Fanuc TP program (LS listing): FM140311.ls

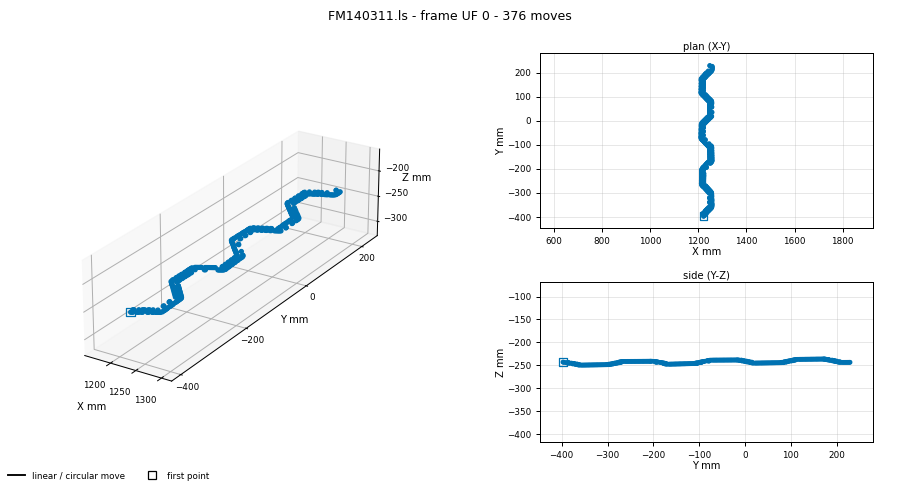
[picture p0: tool path of FM140311.ls in frame UF 0, 376 of 376 moves have a stored position in this frame; points joined in program order, loops and branches not executed]
/PROG  FM140311
/ATTR
OWNER		= MNEDITOR;
COMMENT		= "Auto FANUC move";
PROG_SIZE	= 0;
CREATE		= DATE 26-05-06  TIME 14:03:11;
MODIFIED	= DATE 26-05-06  TIME 14:03:11;
FILE_NAME	= ;
VERSION		= 0;
LINE_COUNT	= 381;
MEMORY_SIZE	= 0;
PROTECT		= READ_WRITE;
TCD:  STACK_SIZE	= 0,
      TASK_PRIORITY	= 50,
      TIME_SLICE	= 0,
      BUSY_LAMP_OFF	= 0,
      ABORT_REQUEST	= 0,
      PAUSE_REQUEST	= 0;
DEFAULT_GROUP	= 1,*,*,*,*;
CONTROL_CODE	= 00000000 00000000;
/MN
   1:  UFRAME_NUM=0 ;
   2:  UTOOL_NUM=1 ;
   3:  R[93]=10 ;
   4:  L P[1] 7mm/sec FINE ;
   5:  L P[2] 7mm/sec CNT50 ;
   6:  L P[3] 7mm/sec CNT50 ;
   7:  L P[4] 7mm/sec CNT50 ;
   8:  L P[5] 7mm/sec CNT50 ;
   9:  L P[6] 7mm/sec CNT50 ;
  10:  L P[7] 7mm/sec CNT50 ;
  11:  L P[8] 7mm/sec CNT50 ;
  12:  L P[9] 7mm/sec CNT50 ;
  13:  L P[10] 7mm/sec CNT50 ;
  14:  L P[11] 7mm/sec CNT50 ;
  15:  L P[12] 7mm/sec CNT50 ;
  16:  L P[13] 7mm/sec CNT50 ;
  17:  L P[14] 7mm/sec CNT50 ;
  18:  L P[15] 7mm/sec CNT50 ;
  19:  L P[16] 7mm/sec CNT50 ;
  20:  L P[17] 7mm/sec CNT50 ;
  21:  L P[18] 7mm/sec CNT50 ;
  22:  L P[19] 7mm/sec CNT50 ;
  23:  L P[20] 7mm/sec CNT50 ;
  24:  L P[21] 7mm/sec CNT50 ;
  25:  L P[22] 7mm/sec CNT50 ;
  26:  L P[23] 7mm/sec CNT50 ;
  27:  L P[24] 7mm/sec CNT50 ;
  28:  L P[25] 7mm/sec CNT50 ;
  29:  L P[26] 7mm/sec CNT50 ;
  30:  L P[27] 7mm/sec CNT50 ;
  31:  L P[28] 7mm/sec CNT50 ;
  32:  L P[29] 7mm/sec CNT50 ;
  33:  L P[30] 7mm/sec CNT50 ;
  34:  L P[31] 7mm/sec CNT50 ;
  35:  L P[32] 7mm/sec CNT50 ;
  36:  L P[33] 7mm/sec CNT50 ;
  37:  L P[34] 7mm/sec CNT50 ;
  38:  L P[35] 7mm/sec CNT50 ;
  39:  L P[36] 7mm/sec CNT50 ;
  40:  L P[37] 7mm/sec CNT50 ;
  41:  L P[38] 7mm/sec CNT50 ;
  42:  L P[39] 7mm/sec CNT50 ;
  43:  L P[40] 7mm/sec CNT50 ;
  44:  L P[41] 7mm/sec CNT50 ;
  45:  L P[42] 7mm/sec CNT50 ;
  46:  L P[43] 7mm/sec CNT50 ;
  47:  L P[44] 7mm/sec CNT50 ;
  48:  L P[45] 7mm/sec CNT50 ;
  49:  L P[46] 7mm/sec CNT50 ;
  50:  L P[47] 7mm/sec CNT50 ;
  51:  L P[48] 7mm/sec CNT50 ;
  52:  L P[49] 7mm/sec CNT50 ;
  53:  L P[50] 7mm/sec CNT50 ;
  54:  L P[51] 7mm/sec CNT50 ;
  55:  L P[52] 7mm/sec CNT50 ;
  56:  L P[53] 7mm/sec CNT50 ;
  57:  L P[54] 7mm/sec CNT50 ;
  58:  L P[55] 7mm/sec CNT50 ;
  59:  L P[56] 7mm/sec CNT50 ;
  60:  L P[57] 7mm/sec CNT50 ;
  61:  L P[58] 7mm/sec CNT50 ;
  62:  L P[59] 7mm/sec CNT50 ;
  63:  L P[60] 7mm/sec CNT50 ;
  64:  L P[61] 7mm/sec CNT50 ;
  65:  L P[62] 7mm/sec CNT50 ;
  66:  L P[63] 7mm/sec CNT50 ;
  67:  L P[64] 7mm/sec CNT50 ;
  68:  L P[65] 7mm/sec CNT50 ;
  69:  L P[66] 7mm/sec CNT50 ;
  70:  L P[67] 7mm/sec CNT50 ;
  71:  L P[68] 7mm/sec CNT50 ;
  72:  L P[69] 7mm/sec CNT50 ;
  73:  L P[70] 7mm/sec CNT50 ;
  74:  L P[71] 7mm/sec CNT50 ;
  75:  L P[72] 7mm/sec CNT50 ;
  76:  L P[73] 7mm/sec CNT50 ;
  77:  L P[74] 7mm/sec CNT50 ;
  78:  L P[75] 7mm/sec CNT50 ;
  79:  L P[76] 7mm/sec CNT50 ;
  80:  L P[77] 7mm/sec CNT50 ;
  81:  L P[78] 7mm/sec CNT50 ;
  82:  L P[79] 7mm/sec CNT50 ;
  83:  L P[80] 7mm/sec CNT50 ;
  84:  L P[81] 7mm/sec CNT50 ;
  85:  L P[82] 7mm/sec CNT50 ;
  86:  L P[83] 7mm/sec CNT50 ;
  87:  L P[84] 7mm/sec CNT50 ;
  88:  L P[85] 7mm/sec CNT50 ;
  89:  L P[86] 7mm/sec CNT50 ;
  90:  L P[87] 7mm/sec CNT50 ;
  91:  L P[88] 7mm/sec CNT50 ;
  92:  L P[89] 7mm/sec CNT50 ;
  93:  L P[90] 7mm/sec CNT50 ;
  94:  L P[91] 7mm/sec CNT50 ;
  95:  L P[92] 7mm/sec CNT50 ;
  96:  L P[93] 7mm/sec CNT50 ;
  97:  L P[94] 7mm/sec CNT50 ;
  98:  L P[95] 7mm/sec CNT50 ;
  99:  L P[96] 7mm/sec CNT50 ;
 100:  L P[97] 7mm/sec CNT50 ;
 101:  L P[98] 7mm/sec CNT50 ;
 102:  L P[99] 7mm/sec CNT50 ;
 103:  L P[100] 7mm/sec CNT50 ;
 104:  L P[101] 7mm/sec CNT50 ;
 105:  L P[102] 7mm/sec CNT50 ;
 106:  L P[103] 7mm/sec CNT50 ;
 107:  L P[104] 7mm/sec CNT50 ;
 108:  L P[105] 7mm/sec CNT50 ;
 109:  L P[106] 7mm/sec CNT50 ;
 110:  L P[107] 7mm/sec CNT50 ;
 111:  L P[108] 7mm/sec CNT50 ;
 112:  L P[109] 7mm/sec CNT50 ;
 113:  L P[110] 7mm/sec CNT50 ;
 114:  L P[111] 7mm/sec CNT50 ;
 115:  L P[112] 7mm/sec CNT50 ;
 116:  L P[113] 7mm/sec CNT50 ;
 117:  L P[114] 7mm/sec CNT50 ;
 118:  L P[115] 7mm/sec CNT50 ;
 119:  L P[116] 7mm/sec CNT50 ;
 120:  L P[117] 7mm/sec CNT50 ;
 121:  L P[118] 7mm/sec CNT50 ;
 122:  L P[119] 7mm/sec CNT50 ;
 123:  L P[120] 7mm/sec CNT50 ;
 124:  L P[121] 7mm/sec CNT50 ;
 125:  L P[122] 7mm/sec CNT50 ;
 126:  L P[123] 7mm/sec CNT50 ;
 127:  L P[124] 7mm/sec CNT50 ;
 128:  L P[125] 7mm/sec CNT50 ;
 129:  L P[126] 7mm/sec CNT50 ;
 130:  L P[127] 7mm/sec CNT50 ;
 131:  L P[128] 7mm/sec CNT50 ;
 132:  L P[129] 7mm/sec CNT50 ;
 133:  L P[130] 7mm/sec CNT50 ;
 134:  L P[131] 7mm/sec CNT50 ;
 135:  L P[132] 7mm/sec CNT50 ;
 136:  L P[133] 7mm/sec CNT50 ;
 137:  L P[134] 7mm/sec CNT50 ;
 138:  L P[135] 7mm/sec CNT50 ;
 139:  L P[136] 7mm/sec CNT50 ;
 140:  L P[137] 7mm/sec CNT50 ;
 141:  L P[138] 7mm/sec CNT50 ;
 142:  L P[139] 7mm/sec CNT50 ;
 143:  L P[140] 7mm/sec CNT50 ;
 144:  L P[141] 7mm/sec CNT50 ;
 145:  L P[142] 7mm/sec CNT50 ;
 146:  L P[143] 7mm/sec CNT50 ;
 147:  L P[144] 7mm/sec CNT50 ;
 148:  L P[145] 7mm/sec CNT50 ;
 149:  L P[146] 7mm/sec CNT50 ;
 150:  L P[147] 7mm/sec CNT50 ;
 151:  L P[148] 7mm/sec CNT50 ;
 152:  L P[149] 7mm/sec CNT50 ;
 153:  L P[150] 7mm/sec CNT50 ;
 154:  L P[151] 7mm/sec CNT50 ;
 155:  L P[152] 7mm/sec CNT50 ;
 156:  L P[153] 7mm/sec CNT50 ;
 157:  L P[154] 7mm/sec CNT50 ;
 158:  L P[155] 7mm/sec CNT50 ;
 159:  L P[156] 7mm/sec CNT50 ;
 160:  L P[157] 7mm/sec CNT50 ;
 161:  L P[158] 7mm/sec CNT50 ;
 162:  L P[159] 7mm/sec CNT50 ;
 163:  L P[160] 7mm/sec CNT50 ;
 164:  L P[161] 7mm/sec CNT50 ;
 165:  L P[162] 7mm/sec CNT50 ;
 166:  L P[163] 7mm/sec CNT50 ;
 167:  L P[164] 7mm/sec CNT50 ;
 168:  L P[165] 7mm/sec CNT50 ;
 169:  L P[166] 7mm/sec CNT50 ;
 170:  L P[167] 7mm/sec CNT50 ;
 171:  L P[168] 7mm/sec CNT50 ;
 172:  L P[169] 7mm/sec CNT50 ;
 173:  L P[170] 7mm/sec CNT50 ;
 174:  L P[171] 7mm/sec CNT50 ;
 175:  L P[172] 7mm/sec CNT50 ;
 176:  L P[173] 7mm/sec CNT50 ;
 177:  L P[174] 7mm/sec CNT50 ;
 178:  L P[175] 7mm/sec CNT50 ;
 179:  L P[176] 7mm/sec CNT50 ;
 180:  L P[177] 7mm/sec CNT50 ;
 181:  L P[178] 7mm/sec CNT50 ;
 182:  L P[179] 7mm/sec CNT50 ;
 183:  L P[180] 7mm/sec CNT50 ;
 184:  L P[181] 7mm/sec CNT50 ;
 185:  L P[182] 7mm/sec CNT50 ;
 186:  L P[183] 7mm/sec CNT50 ;
 187:  L P[184] 7mm/sec CNT50 ;
 188:  L P[185] 7mm/sec CNT50 ;
 189:  L P[186] 7mm/sec CNT50 ;
 190:  L P[187] 7mm/sec CNT50 ;
 191:  L P[188] 7mm/sec CNT50 ;
 192:  L P[189] 7mm/sec CNT50 ;
 193:  L P[190] 7mm/sec CNT50 ;
 194:  L P[191] 7mm/sec CNT50 ;
 195:  L P[192] 7mm/sec CNT50 ;
 196:  L P[193] 7mm/sec CNT50 ;
 197:  L P[194] 7mm/sec CNT50 ;
 198:  L P[195] 7mm/sec CNT50 ;
 199:  L P[196] 7mm/sec CNT50 ;
 200:  L P[197] 7mm/sec CNT50 ;
 201:  L P[198] 7mm/sec CNT50 ;
 202:  L P[199] 7mm/sec CNT50 ;
 203:  L P[200] 7mm/sec CNT50 ;
 204:  L P[201] 7mm/sec CNT50 ;
 205:  L P[202] 7mm/sec CNT50 ;
 206:  L P[203] 7mm/sec CNT50 ;
 207:  L P[204] 7mm/sec CNT50 ;
 208:  L P[205] 7mm/sec CNT50 ;
 209:  L P[206] 7mm/sec CNT50 ;
 210:  L P[207] 7mm/sec CNT50 ;
 211:  L P[208] 7mm/sec CNT50 ;
 212:  L P[209] 7mm/sec CNT50 ;
 213:  L P[210] 7mm/sec CNT50 ;
 214:  L P[211] 7mm/sec CNT50 ;
 215:  L P[212] 7mm/sec CNT50 ;
 216:  L P[213] 7mm/sec CNT50 ;
 217:  L P[214] 7mm/sec CNT50 ;
 218:  L P[215] 7mm/sec CNT50 ;
 219:  L P[216] 7mm/sec CNT50 ;
 220:  L P[217] 7mm/sec CNT50 ;
 221:  L P[218] 7mm/sec CNT50 ;
 222:  L P[219] 7mm/sec CNT50 ;
 223:  L P[220] 7mm/sec CNT50 ;
 224:  L P[221] 7mm/sec CNT50 ;
 225:  L P[222] 7mm/sec CNT50 ;
 226:  L P[223] 7mm/sec CNT50 ;
 227:  L P[224] 7mm/sec CNT50 ;
 228:  L P[225] 7mm/sec CNT50 ;
 229:  L P[226] 7mm/sec CNT50 ;
 230:  L P[227] 7mm/sec CNT50 ;
 231:  L P[228] 7mm/sec CNT50 ;
 232:  L P[229] 7mm/sec CNT50 ;
 233:  L P[230] 7mm/sec CNT50 ;
 234:  L P[231] 7mm/sec CNT50 ;
 235:  L P[232] 7mm/sec CNT50 ;
 236:  L P[233] 7mm/sec CNT50 ;
 237:  L P[234] 7mm/sec CNT50 ;
 238:  L P[235] 7mm/sec CNT50 ;
 239:  L P[236] 7mm/sec CNT50 ;
 240:  L P[237] 7mm/sec CNT50 ;
 241:  L P[238] 7mm/sec CNT50 ;
 242:  L P[239] 7mm/sec CNT50 ;
 243:  L P[240] 7mm/sec CNT50 ;
 244:  L P[241] 7mm/sec CNT50 ;
 245:  L P[242] 7mm/sec CNT50 ;
 246:  L P[243] 7mm/sec CNT50 ;
 247:  L P[244] 7mm/sec CNT50 ;
 248:  L P[245] 7mm/sec CNT50 ;
 249:  L P[246] 7mm/sec CNT50 ;
 250:  L P[247] 7mm/sec CNT50 ;
 251:  L P[248] 7mm/sec CNT50 ;
 252:  L P[249] 7mm/sec CNT50 ;
 253:  L P[250] 7mm/sec CNT50 ;
 254:  L P[251] 7mm/sec CNT50 ;
 255:  L P[252] 7mm/sec CNT50 ;
 256:  L P[253] 7mm/sec CNT50 ;
 257:  L P[254] 7mm/sec CNT50 ;
 258:  L P[255] 7mm/sec CNT50 ;
 259:  L P[256] 7mm/sec CNT50 ;
 260:  L P[257] 7mm/sec CNT50 ;
 261:  L P[258] 7mm/sec CNT50 ;
 262:  L P[259] 7mm/sec CNT50 ;
 263:  L P[260] 7mm/sec CNT50 ;
 264:  L P[261] 7mm/sec CNT50 ;
 265:  L P[262] 7mm/sec CNT50 ;
 266:  L P[263] 7mm/sec CNT50 ;
 267:  L P[264] 7mm/sec CNT50 ;
 268:  L P[265] 7mm/sec CNT50 ;
 269:  L P[266] 7mm/sec CNT50 ;
 270:  L P[267] 7mm/sec CNT50 ;
 271:  L P[268] 7mm/sec CNT50 ;
 272:  L P[269] 7mm/sec CNT50 ;
 273:  L P[270] 7mm/sec CNT50 ;
 274:  L P[271] 7mm/sec CNT50 ;
 275:  L P[272] 7mm/sec CNT50 ;
 276:  L P[273] 7mm/sec CNT50 ;
 277:  L P[274] 7mm/sec CNT50 ;
 278:  L P[275] 7mm/sec CNT50 ;
 279:  L P[276] 7mm/sec CNT50 ;
 280:  L P[277] 7mm/sec CNT50 ;
 281:  L P[278] 7mm/sec CNT50 ;
 282:  L P[279] 7mm/sec CNT50 ;
 283:  L P[280] 7mm/sec CNT50 ;
 284:  L P[281] 7mm/sec CNT50 ;
 285:  L P[282] 7mm/sec CNT50 ;
 286:  L P[283] 7mm/sec CNT50 ;
 287:  L P[284] 7mm/sec CNT50 ;
 288:  L P[285] 7mm/sec CNT50 ;
 289:  L P[286] 7mm/sec CNT50 ;
 290:  L P[287] 7mm/sec CNT50 ;
 291:  L P[288] 7mm/sec CNT50 ;
 292:  L P[289] 7mm/sec CNT50 ;
 293:  L P[290] 7mm/sec CNT50 ;
 294:  L P[291] 7mm/sec CNT50 ;
 295:  L P[292] 7mm/sec CNT50 ;
 296:  L P[293] 7mm/sec CNT50 ;
 297:  L P[294] 7mm/sec CNT50 ;
 298:  L P[295] 7mm/sec CNT50 ;
 299:  L P[296] 7mm/sec CNT50 ;
 300:  L P[297] 7mm/sec CNT50 ;
 301:  L P[298] 7mm/sec CNT50 ;
 302:  L P[299] 7mm/sec CNT50 ;
 303:  L P[300] 7mm/sec CNT50 ;
 304:  L P[301] 7mm/sec CNT50 ;
 305:  L P[302] 7mm/sec CNT50 ;
 306:  L P[303] 7mm/sec CNT50 ;
 307:  L P[304] 7mm/sec CNT50 ;
 308:  L P[305] 7mm/sec CNT50 ;
 309:  L P[306] 7mm/sec CNT50 ;
 310:  L P[307] 7mm/sec CNT50 ;
 311:  L P[308] 7mm/sec CNT50 ;
 312:  L P[309] 7mm/sec CNT50 ;
 313:  L P[310] 7mm/sec CNT50 ;
 314:  L P[311] 7mm/sec CNT50 ;
 315:  L P[312] 7mm/sec CNT50 ;
 316:  L P[313] 7mm/sec CNT50 ;
 317:  L P[314] 7mm/sec CNT50 ;
 318:  L P[315] 7mm/sec CNT50 ;
 319:  L P[316] 7mm/sec CNT50 ;
 320:  L P[317] 7mm/sec CNT50 ;
 321:  L P[318] 7mm/sec CNT50 ;
 322:  L P[319] 7mm/sec CNT50 ;
 323:  L P[320] 7mm/sec CNT50 ;
 324:  L P[321] 7mm/sec CNT50 ;
 325:  L P[322] 7mm/sec CNT50 ;
 326:  L P[323] 7mm/sec CNT50 ;
 327:  L P[324] 7mm/sec CNT50 ;
 328:  L P[325] 7mm/sec CNT50 ;
 329:  L P[326] 7mm/sec CNT50 ;
 330:  L P[327] 7mm/sec CNT50 ;
 331:  L P[328] 7mm/sec CNT50 ;
 332:  L P[329] 7mm/sec CNT50 ;
 333:  L P[330] 7mm/sec CNT50 ;
 334:  L P[331] 7mm/sec CNT50 ;
 335:  L P[332] 7mm/sec CNT50 ;
 336:  L P[333] 7mm/sec CNT50 ;
 337:  L P[334] 7mm/sec CNT50 ;
 338:  L P[335] 7mm/sec CNT50 ;
 339:  L P[336] 7mm/sec CNT50 ;
 340:  L P[337] 7mm/sec CNT50 ;
 341:  L P[338] 7mm/sec CNT50 ;
 342:  L P[339] 7mm/sec CNT50 ;
 343:  L P[340] 7mm/sec CNT50 ;
 344:  L P[341] 7mm/sec CNT50 ;
 345:  L P[342] 7mm/sec CNT50 ;
 346:  L P[343] 7mm/sec CNT50 ;
 347:  L P[344] 7mm/sec CNT50 ;
 348:  L P[345] 7mm/sec CNT50 ;
 349:  L P[346] 7mm/sec CNT50 ;
 350:  L P[347] 7mm/sec CNT50 ;
 351:  L P[348] 7mm/sec CNT50 ;
 352:  L P[349] 7mm/sec CNT50 ;
 353:  L P[350] 7mm/sec CNT50 ;
 354:  L P[351] 7mm/sec CNT50 ;
 355:  L P[352] 7mm/sec CNT50 ;
 356:  L P[353] 7mm/sec CNT50 ;
 357:  L P[354] 7mm/sec CNT50 ;
 358:  L P[355] 7mm/sec CNT50 ;
 359:  L P[356] 7mm/sec CNT50 ;
 360:  L P[357] 7mm/sec CNT50 ;
 361:  L P[358] 7mm/sec CNT50 ;
 362:  L P[359] 7mm/sec CNT50 ;
 363:  L P[360] 7mm/sec CNT50 ;
 364:  L P[361] 7mm/sec CNT50 ;
 365:  L P[362] 7mm/sec CNT50 ;
 366:  L P[363] 7mm/sec CNT50 ;
 367:  L P[364] 7mm/sec CNT50 ;
 368:  L P[365] 7mm/sec CNT50 ;
 369:  L P[366] 7mm/sec CNT50 ;
 370:  L P[367] 7mm/sec CNT50 ;
 371:  L P[368] 7mm/sec CNT50 ;
 372:  L P[369] 7mm/sec CNT50 ;
 373:  L P[370] 7mm/sec CNT50 ;
 374:  L P[371] 7mm/sec CNT50 ;
 375:  L P[372] 7mm/sec CNT50 ;
 376:  L P[373] 7mm/sec CNT50 ;
 377:  L P[374] 7mm/sec CNT50 ;
 378:  L P[375] 7mm/sec CNT50 ;
 379:  L P[376] 7mm/sec FINE ;
 380:  R[93]=1 ;
 381:  END ;
/POS
P[1]{
   GP1:
	UF : 0, UT : 1,		CONFIG : 'N U T, 0, 0, 0',
	X = 1221.690  mm,	Y = -397.242  mm,	Z = -243.032  mm,
	W = 0.000 deg,	P = 30.000 deg,	R = 137.115 deg
};
P[2]{
   GP1:
	UF : 0, UT : 1,		CONFIG : 'N U T, 0, 0, 0',
	X = 1223.040  mm,	Y = -395.790  mm,	Z = -243.294  mm,
	W = 0.000 deg,	P = 30.000 deg,	R = 137.115 deg
};
P[3]{
   GP1:
	UF : 0, UT : 1,		CONFIG : 'N U T, 0, 0, 0',
	X = 1224.389  mm,	Y = -394.337  mm,	Z = -243.556  mm,
	W = 0.000 deg,	P = 30.000 deg,	R = 137.115 deg
};
P[4]{
   GP1:
	UF : 0, UT : 1,		CONFIG : 'N U T, 0, 0, 0',
	X = 1218.411  mm,	Y = -386.079  mm,	Z = -243.818  mm,
	W = 0.000 deg,	P = 30.000 deg,	R = 137.115 deg
};
P[5]{
   GP1:
	UF : 0, UT : 1,		CONFIG : 'N U T, 0, 0, 0',
	X = 1219.760  mm,	Y = -384.626  mm,	Z = -244.080  mm,
	W = 0.000 deg,	P = 30.000 deg,	R = 137.115 deg
};
P[6]{
   GP1:
	UF : 0, UT : 1,		CONFIG : 'N U T, 0, 0, 0',
	X = 1228.437  mm,	Y = -389.978  mm,	Z = -244.342  mm,
	W = 0.000 deg,	P = 30.000 deg,	R = 137.115 deg
};
P[7]{
   GP1:
	UF : 0, UT : 1,		CONFIG : 'N U T, 0, 0, 0',
	X = 1229.786  mm,	Y = -388.526  mm,	Z = -244.604  mm,
	W = 0.000 deg,	P = 30.000 deg,	R = 137.115 deg
};
P[8]{
   GP1:
	UF : 0, UT : 1,		CONFIG : 'N U T, 0, 0, 0',
	X = 1231.136  mm,	Y = -387.073  mm,	Z = -244.866  mm,
	W = 0.000 deg,	P = 30.000 deg,	R = 137.115 deg
};
P[9]{
   GP1:
	UF : 0, UT : 1,		CONFIG : 'N U T, 0, 0, 0',
	X = 1225.158  mm,	Y = -378.815  mm,	Z = -245.128  mm,
	W = 0.000 deg,	P = 30.000 deg,	R = 137.115 deg
};
P[10]{
   GP1:
	UF : 0, UT : 1,		CONFIG : 'N U T, 0, 0, 0',
	X = 1233.834  mm,	Y = -384.167  mm,	Z = -245.390  mm,
	W = 0.000 deg,	P = 30.000 deg,	R = 137.115 deg
};
P[11]{
   GP1:
	UF : 0, UT : 1,		CONFIG : 'N U T, 0, 0, 0',
	X = 1235.184  mm,	Y = -382.714  mm,	Z = -245.652  mm,
	W = 0.000 deg,	P = 30.000 deg,	R = 137.115 deg
};
P[12]{
   GP1:
	UF : 0, UT : 1,		CONFIG : 'N U T, 0, 0, 0',
	X = 1229.206  mm,	Y = -374.456  mm,	Z = -245.914  mm,
	W = 0.000 deg,	P = 30.000 deg,	R = 137.115 deg
};
P[13]{
   GP1:
	UF : 0, UT : 1,		CONFIG : 'N U T, 0, 0, 0',
	X = 1230.555  mm,	Y = -373.003  mm,	Z = -246.176  mm,
	W = 0.000 deg,	P = 30.000 deg,	R = 137.115 deg
};
P[14]{
   GP1:
	UF : 0, UT : 1,		CONFIG : 'N U T, 0, 0, 0',
	X = 1231.904  mm,	Y = -371.551  mm,	Z = -246.438  mm,
	W = 0.000 deg,	P = 30.000 deg,	R = 137.115 deg
};
P[15]{
   GP1:
	UF : 0, UT : 1,		CONFIG : 'N U T, 0, 0, 0',
	X = 1240.581  mm,	Y = -376.903  mm,	Z = -246.700  mm,
	W = 0.000 deg,	P = 30.000 deg,	R = 137.115 deg
};
P[16]{
   GP1:
	UF : 0, UT : 1,		CONFIG : 'N U T, 0, 0, 0',
	X = 1241.930  mm,	Y = -375.450  mm,	Z = -246.962  mm,
	W = 0.000 deg,	P = 30.000 deg,	R = 137.115 deg
};
P[17]{
   GP1:
	UF : 0, UT : 1,		CONFIG : 'N U T, 0, 0, 0',
	X = 1235.952  mm,	Y = -367.192  mm,	Z = -247.224  mm,
	W = 0.000 deg,	P = 30.000 deg,	R = 137.115 deg
};
P[18]{
   GP1:
	UF : 0, UT : 1,		CONFIG : 'N U T, 0, 0, 0',
	X = 1237.302  mm,	Y = -365.739  mm,	Z = -247.486  mm,
	W = 0.000 deg,	P = 30.000 deg,	R = 137.115 deg
};
P[19]{
   GP1:
	UF : 0, UT : 1,		CONFIG : 'N U T, 0, 0, 0',
	X = 1245.978  mm,	Y = -371.092  mm,	Z = -247.748  mm,
	W = 0.000 deg,	P = 30.000 deg,	R = 137.115 deg
};
P[20]{
   GP1:
	UF : 0, UT : 1,		CONFIG : 'N U T, 0, 0, 0',
	X = 1247.328  mm,	Y = -369.639  mm,	Z = -248.010  mm,
	W = 0.000 deg,	P = 30.000 deg,	R = 137.115 deg
};
P[21]{
   GP1:
	UF : 0, UT : 1,		CONFIG : 'N U T, 0, 0, 0',
	X = 1241.350  mm,	Y = -361.381  mm,	Z = -248.271  mm,
	W = 0.000 deg,	P = 30.000 deg,	R = 137.115 deg
};
P[22]{
   GP1:
	UF : 0, UT : 1,		CONFIG : 'N U T, 0, 0, 0',
	X = 1250.026  mm,	Y = -366.733  mm,	Z = -248.533  mm,
	W = 0.000 deg,	P = 30.000 deg,	R = 145.950 deg
};
P[23]{
   GP1:
	UF : 0, UT : 1,		CONFIG : 'N U T, 0, 0, 0',
	X = 1251.376  mm,	Y = -365.280  mm,	Z = -248.795  mm,
	W = 0.000 deg,	P = 30.000 deg,	R = 154.785 deg
};
P[24]{
   GP1:
	UF : 0, UT : 1,		CONFIG : 'N U T, 0, 0, 0',
	X = 1252.725  mm,	Y = -363.828  mm,	Z = -249.057  mm,
	W = 0.000 deg,	P = 30.000 deg,	R = 163.620 deg
};
P[25]{
   GP1:
	UF : 0, UT : 1,		CONFIG : 'N U T, 0, 0, 0',
	X = 1254.074  mm,	Y = -362.375  mm,	Z = -249.319  mm,
	W = 0.000 deg,	P = 30.000 deg,	R = 172.455 deg
};
P[26]{
   GP1:
	UF : 0, UT : 1,		CONFIG : 'N U T, 0, 0, 0',
	X = 1255.424  mm,	Y = -360.922  mm,	Z = -249.581  mm,
	W = 0.000 deg,	P = 30.000 deg,	R = -178.709 deg
};
P[27]{
   GP1:
	UF : 0, UT : 1,		CONFIG : 'N U T, 0, 0, 0',
	X = 1256.911  mm,	Y = -357.658  mm,	Z = -249.612  mm,
	W = 0.000 deg,	P = 30.000 deg,	R = -178.709 deg
};
P[28]{
   GP1:
	UF : 0, UT : 1,		CONFIG : 'N U T, 0, 0, 0',
	X = 1246.882  mm,	Y = -355.698  mm,	Z = -249.584  mm,
	W = 0.000 deg,	P = 30.000 deg,	R = -178.709 deg
};
P[29]{
   GP1:
	UF : 0, UT : 1,		CONFIG : 'N U T, 0, 0, 0',
	X = 1256.834  mm,	Y = -353.473  mm,	Z = -249.552  mm,
	W = 0.000 deg,	P = 30.000 deg,	R = -178.709 deg
};
P[30]{
   GP1:
	UF : 0, UT : 1,		CONFIG : 'N U T, 0, 0, 0',
	X = 1256.789  mm,	Y = -351.474  mm,	Z = -249.520  mm,
	W = 0.000 deg,	P = 30.000 deg,	R = -178.709 deg
};
P[31]{
   GP1:
	UF : 0, UT : 1,		CONFIG : 'N U T, 0, 0, 0',
	X = 1256.744  mm,	Y = -349.475  mm,	Z = -249.488  mm,
	W = 0.000 deg,	P = 30.000 deg,	R = -178.709 deg
};
P[32]{
   GP1:
	UF : 0, UT : 1,		CONFIG : 'N U T, 0, 0, 0',
	X = 1256.699  mm,	Y = -347.476  mm,	Z = -249.455  mm,
	W = 0.000 deg,	P = 30.000 deg,	R = -178.709 deg
};
P[33]{
   GP1:
	UF : 0, UT : 1,		CONFIG : 'N U T, 0, 0, 0',
	X = 1256.654  mm,	Y = -345.476  mm,	Z = -249.423  mm,
	W = 0.000 deg,	P = 30.000 deg,	R = -178.709 deg
};
P[34]{
   GP1:
	UF : 0, UT : 1,		CONFIG : 'N U T, 0, 0, 0',
	X = 1256.609  mm,	Y = -343.477  mm,	Z = -249.391  mm,
	W = 0.000 deg,	P = 30.000 deg,	R = -178.709 deg
};
P[35]{
   GP1:
	UF : 0, UT : 1,		CONFIG : 'N U T, 0, 0, 0',
	X = 1256.564  mm,	Y = -341.478  mm,	Z = -249.359  mm,
	W = 0.000 deg,	P = 30.000 deg,	R = -178.709 deg
};
P[36]{
   GP1:
	UF : 0, UT : 1,		CONFIG : 'N U T, 0, 0, 0',
	X = 1246.522  mm,	Y = -339.704  mm,	Z = -249.327  mm,
	W = 0.000 deg,	P = 30.000 deg,	R = -178.709 deg
};
P[37]{
   GP1:
	UF : 0, UT : 1,		CONFIG : 'N U T, 0, 0, 0',
	X = 1246.477  mm,	Y = -337.705  mm,	Z = -249.294  mm,
	W = 0.000 deg,	P = 30.000 deg,	R = -178.709 deg
};
P[38]{
   GP1:
	UF : 0, UT : 1,		CONFIG : 'N U T, 0, 0, 0',
	X = 1256.429  mm,	Y = -335.480  mm,	Z = -249.262  mm,
	W = 0.000 deg,	P = 30.000 deg,	R = -178.709 deg
};
P[39]{
   GP1:
	UF : 0, UT : 1,		CONFIG : 'N U T, 0, 0, 0',
	X = 1256.384  mm,	Y = -333.481  mm,	Z = -249.230  mm,
	W = 0.000 deg,	P = 30.000 deg,	R = -178.709 deg
};
P[40]{
   GP1:
	UF : 0, UT : 1,		CONFIG : 'N U T, 0, 0, 0',
	X = 1256.339  mm,	Y = -331.482  mm,	Z = -249.198  mm,
	W = 0.000 deg,	P = 30.000 deg,	R = -178.709 deg
};
P[41]{
   GP1:
	UF : 0, UT : 1,		CONFIG : 'N U T, 0, 0, 0',
	X = 1256.294  mm,	Y = -329.482  mm,	Z = -249.166  mm,
	W = 0.000 deg,	P = 30.000 deg,	R = -178.709 deg
};
P[42]{
   GP1:
	UF : 0, UT : 1,		CONFIG : 'N U T, 0, 0, 0',
	X = 1256.249  mm,	Y = -327.483  mm,	Z = -249.134  mm,
	W = 0.000 deg,	P = 30.000 deg,	R = -178.709 deg
};
P[43]{
   GP1:
	UF : 0, UT : 1,		CONFIG : 'N U T, 0, 0, 0',
	X = 1256.204  mm,	Y = -325.484  mm,	Z = -249.101  mm,
	W = 0.000 deg,	P = 30.000 deg,	R = -178.709 deg
};
P[44]{
   GP1:
	UF : 0, UT : 1,		CONFIG : 'N U T, 0, 0, 0',
	X = 1256.159  mm,	Y = -323.485  mm,	Z = -249.069  mm,
	W = 0.000 deg,	P = 30.000 deg,	R = -178.709 deg
};
P[45]{
   GP1:
	UF : 0, UT : 1,		CONFIG : 'N U T, 0, 0, 0',
	X = 1246.116  mm,	Y = -321.711  mm,	Z = -249.037  mm,
	W = 0.000 deg,	P = 30.000 deg,	R = -178.709 deg
};
P[46]{
   GP1:
	UF : 0, UT : 1,		CONFIG : 'N U T, 0, 0, 0',
	X = 1246.071  mm,	Y = -319.712  mm,	Z = -249.005  mm,
	W = 0.000 deg,	P = 30.000 deg,	R = -178.709 deg
};
P[47]{
   GP1:
	UF : 0, UT : 1,		CONFIG : 'N U T, 0, 0, 0',
	X = 1256.024  mm,	Y = -317.487  mm,	Z = -248.973  mm,
	W = 0.000 deg,	P = 30.000 deg,	R = -178.709 deg
};
P[48]{
   GP1:
	UF : 0, UT : 1,		CONFIG : 'N U T, 0, 0, 0',
	X = 1255.979  mm,	Y = -315.488  mm,	Z = -248.941  mm,
	W = 0.000 deg,	P = 30.000 deg,	R = -178.709 deg
};
P[49]{
   GP1:
	UF : 0, UT : 1,		CONFIG : 'N U T, 0, 0, 0',
	X = 1255.934  mm,	Y = -313.489  mm,	Z = -248.908  mm,
	W = 0.000 deg,	P = 30.000 deg,	R = -178.709 deg
};
P[50]{
   GP1:
	UF : 0, UT : 1,		CONFIG : 'N U T, 0, 0, 0',
	X = 1255.889  mm,	Y = -311.489  mm,	Z = -248.876  mm,
	W = 0.000 deg,	P = 30.000 deg,	R = -178.709 deg
};
P[51]{
   GP1:
	UF : 0, UT : 1,		CONFIG : 'N U T, 0, 0, 0',
	X = 1255.844  mm,	Y = -309.490  mm,	Z = -248.844  mm,
	W = 0.000 deg,	P = 30.000 deg,	R = -171.526 deg
};
P[52]{
   GP1:
	UF : 0, UT : 1,		CONFIG : 'N U T, 0, 0, 0',
	X = 1255.799  mm,	Y = -307.491  mm,	Z = -248.812  mm,
	W = 0.000 deg,	P = 30.000 deg,	R = -163.372 deg
};
P[53]{
   GP1:
	UF : 0, UT : 1,		CONFIG : 'N U T, 0, 0, 0',
	X = 1255.754  mm,	Y = -305.492  mm,	Z = -248.780  mm,
	W = 0.000 deg,	P = 30.000 deg,	R = -155.219 deg
};
P[54]{
   GP1:
	UF : 0, UT : 1,		CONFIG : 'N U T, 0, 0, 0',
	X = 1255.709  mm,	Y = -303.492  mm,	Z = -248.747  mm,
	W = 0.000 deg,	P = 30.000 deg,	R = -147.065 deg
};
P[55]{
   GP1:
	UF : 0, UT : 1,		CONFIG : 'N U T, 0, 0, 0',
	X = 1255.663  mm,	Y = -301.493  mm,	Z = -248.715  mm,
	W = 0.000 deg,	P = 30.000 deg,	R = -138.912 deg
};
P[56]{
   GP1:
	UF : 0, UT : 1,		CONFIG : 'N U T, 0, 0, 0',
	X = 1255.542  mm,	Y = -299.157  mm,	Z = -248.691  mm,
	W = 0.000 deg,	P = 30.000 deg,	R = -137.942 deg
};
P[57]{
   GP1:
	UF : 0, UT : 1,		CONFIG : 'N U T, 0, 0, 0',
	X = 1254.021  mm,	Y = -296.386  mm,	Z = -248.621  mm,
	W = 0.000 deg,	P = 30.000 deg,	R = -137.942 deg
};
P[58]{
   GP1:
	UF : 0, UT : 1,		CONFIG : 'N U T, 0, 0, 0',
	X = 1245.270  mm,	Y = -301.615  mm,	Z = -248.335  mm,
	W = 0.000 deg,	P = 30.000 deg,	R = -137.942 deg
};
P[59]{
   GP1:
	UF : 0, UT : 1,		CONFIG : 'N U T, 0, 0, 0',
	X = 1251.369  mm,	Y = -293.447  mm,	Z = -248.048  mm,
	W = 0.000 deg,	P = 30.000 deg,	R = -137.942 deg
};
P[60]{
   GP1:
	UF : 0, UT : 1,		CONFIG : 'N U T, 0, 0, 0',
	X = 1250.043  mm,	Y = -291.977  mm,	Z = -247.762  mm,
	W = 0.000 deg,	P = 30.000 deg,	R = -137.942 deg
};
P[61]{
   GP1:
	UF : 0, UT : 1,		CONFIG : 'N U T, 0, 0, 0',
	X = 1241.292  mm,	Y = -297.206  mm,	Z = -247.475  mm,
	W = 0.000 deg,	P = 30.000 deg,	R = -137.942 deg
};
P[62]{
   GP1:
	UF : 0, UT : 1,		CONFIG : 'N U T, 0, 0, 0',
	X = 1247.391  mm,	Y = -289.038  mm,	Z = -247.189  mm,
	W = 0.000 deg,	P = 30.000 deg,	R = -137.942 deg
};
P[63]{
   GP1:
	UF : 0, UT : 1,		CONFIG : 'N U T, 0, 0, 0',
	X = 1246.065  mm,	Y = -287.568  mm,	Z = -246.902  mm,
	W = 0.000 deg,	P = 30.000 deg,	R = -137.942 deg
};
P[64]{
   GP1:
	UF : 0, UT : 1,		CONFIG : 'N U T, 0, 0, 0',
	X = 1237.314  mm,	Y = -292.797  mm,	Z = -246.616  mm,
	W = 0.000 deg,	P = 30.000 deg,	R = -137.942 deg
};
P[65]{
   GP1:
	UF : 0, UT : 1,		CONFIG : 'N U T, 0, 0, 0',
	X = 1243.413  mm,	Y = -284.629  mm,	Z = -246.329  mm,
	W = 0.000 deg,	P = 30.000 deg,	R = -137.942 deg
};
P[66]{
   GP1:
	UF : 0, UT : 1,		CONFIG : 'N U T, 0, 0, 0',
	X = 1242.087  mm,	Y = -283.159  mm,	Z = -246.042  mm,
	W = 0.000 deg,	P = 30.000 deg,	R = -137.942 deg
};
P[67]{
   GP1:
	UF : 0, UT : 1,		CONFIG : 'N U T, 0, 0, 0',
	X = 1233.337  mm,	Y = -288.389  mm,	Z = -245.756  mm,
	W = 0.000 deg,	P = 30.000 deg,	R = -137.942 deg
};
P[68]{
   GP1:
	UF : 0, UT : 1,		CONFIG : 'N U T, 0, 0, 0',
	X = 1239.435  mm,	Y = -280.220  mm,	Z = -245.469  mm,
	W = 0.000 deg,	P = 30.000 deg,	R = -137.942 deg
};
P[69]{
   GP1:
	UF : 0, UT : 1,		CONFIG : 'N U T, 0, 0, 0',
	X = 1238.109  mm,	Y = -278.750  mm,	Z = -245.183  mm,
	W = 0.000 deg,	P = 30.000 deg,	R = -137.942 deg
};
P[70]{
   GP1:
	UF : 0, UT : 1,		CONFIG : 'N U T, 0, 0, 0',
	X = 1229.359  mm,	Y = -283.980  mm,	Z = -244.896  mm,
	W = 0.000 deg,	P = 30.000 deg,	R = -137.942 deg
};
P[71]{
   GP1:
	UF : 0, UT : 1,		CONFIG : 'N U T, 0, 0, 0',
	X = 1235.458  mm,	Y = -275.811  mm,	Z = -244.610  mm,
	W = 0.000 deg,	P = 30.000 deg,	R = -137.942 deg
};
P[72]{
   GP1:
	UF : 0, UT : 1,		CONFIG : 'N U T, 0, 0, 0',
	X = 1234.132  mm,	Y = -274.342  mm,	Z = -244.323  mm,
	W = 0.000 deg,	P = 30.000 deg,	R = -137.942 deg
};
P[73]{
   GP1:
	UF : 0, UT : 1,		CONFIG : 'N U T, 0, 0, 0',
	X = 1225.381  mm,	Y = -279.571  mm,	Z = -244.037  mm,
	W = 0.000 deg,	P = 30.000 deg,	R = -137.942 deg
};
P[74]{
   GP1:
	UF : 0, UT : 1,		CONFIG : 'N U T, 0, 0, 0',
	X = 1231.480  mm,	Y = -271.402  mm,	Z = -243.750  mm,
	W = 0.000 deg,	P = 30.000 deg,	R = -137.942 deg
};
P[75]{
   GP1:
	UF : 0, UT : 1,		CONFIG : 'N U T, 0, 0, 0',
	X = 1230.154  mm,	Y = -269.933  mm,	Z = -243.464  mm,
	W = 0.000 deg,	P = 30.000 deg,	R = -137.942 deg
};
P[76]{
   GP1:
	UF : 0, UT : 1,		CONFIG : 'N U T, 0, 0, 0',
	X = 1221.403  mm,	Y = -275.162  mm,	Z = -243.177  mm,
	W = 0.000 deg,	P = 30.000 deg,	R = -137.942 deg
};
P[77]{
   GP1:
	UF : 0, UT : 1,		CONFIG : 'N U T, 0, 0, 0',
	X = 1220.077  mm,	Y = -273.692  mm,	Z = -242.891  mm,
	W = 0.000 deg,	P = 30.000 deg,	R = -140.044 deg
};
P[78]{
   GP1:
	UF : 0, UT : 1,		CONFIG : 'N U T, 0, 0, 0',
	X = 1218.751  mm,	Y = -272.223  mm,	Z = -242.604  mm,
	W = 0.000 deg,	P = 30.000 deg,	R = -148.694 deg
};
P[79]{
   GP1:
	UF : 0, UT : 1,		CONFIG : 'N U T, 0, 0, 0',
	X = 1217.425  mm,	Y = -270.753  mm,	Z = -242.318  mm,
	W = 0.000 deg,	P = 30.000 deg,	R = -157.343 deg
};
P[80]{
   GP1:
	UF : 0, UT : 1,		CONFIG : 'N U T, 0, 0, 0',
	X = 1216.099  mm,	Y = -269.284  mm,	Z = -242.031  mm,
	W = 0.000 deg,	P = 30.000 deg,	R = -165.993 deg
};
P[81]{
   GP1:
	UF : 0, UT : 1,		CONFIG : 'N U T, 0, 0, 0',
	X = 1214.773  mm,	Y = -267.814  mm,	Z = -241.744  mm,
	W = 0.000 deg,	P = 30.000 deg,	R = -174.643 deg
};
P[82]{
   GP1:
	UF : 0, UT : 1,		CONFIG : 'N U T, 0, 0, 0',
	X = 1213.299  mm,	Y = -266.130  mm,	Z = -241.504  mm,
	W = 0.000 deg,	P = 30.000 deg,	R = 178.809 deg
};
P[83]{
   GP1:
	UF : 0, UT : 1,		CONFIG : 'N U T, 0, 0, 0',
	X = 1222.378  mm,	Y = -263.014  mm,	Z = -241.502  mm,
	W = 0.000 deg,	P = 30.000 deg,	R = 178.809 deg
};
P[84]{
   GP1:
	UF : 0, UT : 1,		CONFIG : 'N U T, 0, 0, 0',
	X = 1212.422  mm,	Y = -260.806  mm,	Z = -241.490  mm,
	W = 0.000 deg,	P = 30.000 deg,	R = 178.809 deg
};
P[85]{
   GP1:
	UF : 0, UT : 1,		CONFIG : 'N U T, 0, 0, 0',
	X = 1212.464  mm,	Y = -258.807  mm,	Z = -241.479  mm,
	W = 0.000 deg,	P = 30.000 deg,	R = 178.809 deg
};
P[86]{
   GP1:
	UF : 0, UT : 1,		CONFIG : 'N U T, 0, 0, 0',
	X = 1222.503  mm,	Y = -257.015  mm,	Z = -241.467  mm,
	W = 0.000 deg,	P = 30.000 deg,	R = 178.809 deg
};
P[87]{
   GP1:
	UF : 0, UT : 1,		CONFIG : 'N U T, 0, 0, 0',
	X = 1222.545  mm,	Y = -255.016  mm,	Z = -241.455  mm,
	W = 0.000 deg,	P = 30.000 deg,	R = 178.809 deg
};
P[88]{
   GP1:
	UF : 0, UT : 1,		CONFIG : 'N U T, 0, 0, 0',
	X = 1222.586  mm,	Y = -253.016  mm,	Z = -241.443  mm,
	W = 0.000 deg,	P = 30.000 deg,	R = 178.809 deg
};
P[89]{
   GP1:
	UF : 0, UT : 1,		CONFIG : 'N U T, 0, 0, 0',
	X = 1212.630  mm,	Y = -250.809  mm,	Z = -241.432  mm,
	W = 0.000 deg,	P = 30.000 deg,	R = 178.809 deg
};
P[90]{
   GP1:
	UF : 0, UT : 1,		CONFIG : 'N U T, 0, 0, 0',
	X = 1212.671  mm,	Y = -248.809  mm,	Z = -241.420  mm,
	W = 0.000 deg,	P = 30.000 deg,	R = 178.809 deg
};
P[91]{
   GP1:
	UF : 0, UT : 1,		CONFIG : 'N U T, 0, 0, 0',
	X = 1222.711  mm,	Y = -247.017  mm,	Z = -241.408  mm,
	W = 0.000 deg,	P = 30.000 deg,	R = 178.809 deg
};
P[92]{
   GP1:
	UF : 0, UT : 1,		CONFIG : 'N U T, 0, 0, 0',
	X = 1222.752  mm,	Y = -245.018  mm,	Z = -241.396  mm,
	W = 0.000 deg,	P = 30.000 deg,	R = 178.809 deg
};
P[93]{
   GP1:
	UF : 0, UT : 1,		CONFIG : 'N U T, 0, 0, 0',
	X = 1212.796  mm,	Y = -242.811  mm,	Z = -241.385  mm,
	W = 0.000 deg,	P = 30.000 deg,	R = 178.809 deg
};
P[94]{
   GP1:
	UF : 0, UT : 1,		CONFIG : 'N U T, 0, 0, 0',
	X = 1212.838  mm,	Y = -240.811  mm,	Z = -241.373  mm,
	W = 0.000 deg,	P = 30.000 deg,	R = 178.809 deg
};
P[95]{
   GP1:
	UF : 0, UT : 1,		CONFIG : 'N U T, 0, 0, 0',
	X = 1222.877  mm,	Y = -239.019  mm,	Z = -241.361  mm,
	W = 0.000 deg,	P = 30.000 deg,	R = 178.809 deg
};
P[96]{
   GP1:
	UF : 0, UT : 1,		CONFIG : 'N U T, 0, 0, 0',
	X = 1222.919  mm,	Y = -237.020  mm,	Z = -241.349  mm,
	W = 0.000 deg,	P = 30.000 deg,	R = 178.809 deg
};
P[97]{
   GP1:
	UF : 0, UT : 1,		CONFIG : 'N U T, 0, 0, 0',
	X = 1212.962  mm,	Y = -234.812  mm,	Z = -241.338  mm,
	W = 0.000 deg,	P = 30.000 deg,	R = 178.809 deg
};
P[98]{
   GP1:
	UF : 0, UT : 1,		CONFIG : 'N U T, 0, 0, 0',
	X = 1213.004  mm,	Y = -232.813  mm,	Z = -241.326  mm,
	W = 0.000 deg,	P = 30.000 deg,	R = 178.809 deg
};
P[99]{
   GP1:
	UF : 0, UT : 1,		CONFIG : 'N U T, 0, 0, 0',
	X = 1223.043  mm,	Y = -231.021  mm,	Z = -241.314  mm,
	W = 0.000 deg,	P = 30.000 deg,	R = 178.809 deg
};
P[100]{
   GP1:
	UF : 0, UT : 1,		CONFIG : 'N U T, 0, 0, 0',
	X = 1223.085  mm,	Y = -229.022  mm,	Z = -241.302  mm,
	W = 0.000 deg,	P = 30.000 deg,	R = 178.809 deg
};
P[101]{
   GP1:
	UF : 0, UT : 1,		CONFIG : 'N U T, 0, 0, 0',
	X = 1223.126  mm,	Y = -227.022  mm,	Z = -241.291  mm,
	W = 0.000 deg,	P = 30.000 deg,	R = 178.809 deg
};
P[102]{
   GP1:
	UF : 0, UT : 1,		CONFIG : 'N U T, 0, 0, 0',
	X = 1213.170  mm,	Y = -224.815  mm,	Z = -241.279  mm,
	W = 0.000 deg,	P = 30.000 deg,	R = 178.809 deg
};
P[103]{
   GP1:
	UF : 0, UT : 1,		CONFIG : 'N U T, 0, 0, 0',
	X = 1213.212  mm,	Y = -222.815  mm,	Z = -241.267  mm,
	W = 0.000 deg,	P = 30.000 deg,	R = 178.809 deg
};
P[104]{
   GP1:
	UF : 0, UT : 1,		CONFIG : 'N U T, 0, 0, 0',
	X = 1223.251  mm,	Y = -221.023  mm,	Z = -241.255  mm,
	W = 0.000 deg,	P = 30.000 deg,	R = 178.809 deg
};
P[105]{
   GP1:
	UF : 0, UT : 1,		CONFIG : 'N U T, 0, 0, 0',
	X = 1223.293  mm,	Y = -219.024  mm,	Z = -241.244  mm,
	W = 0.000 deg,	P = 30.000 deg,	R = 178.809 deg
};
P[106]{
   GP1:
	UF : 0, UT : 1,		CONFIG : 'N U T, 0, 0, 0',
	X = 1213.336  mm,	Y = -216.817  mm,	Z = -241.232  mm,
	W = 0.000 deg,	P = 30.000 deg,	R = 178.809 deg
};
P[107]{
   GP1:
	UF : 0, UT : 1,		CONFIG : 'N U T, 0, 0, 0',
	X = 1213.378  mm,	Y = -214.817  mm,	Z = -241.220  mm,
	W = 0.000 deg,	P = 30.000 deg,	R = 178.809 deg
};
P[108]{
   GP1:
	UF : 0, UT : 1,		CONFIG : 'N U T, 0, 0, 0',
	X = 1213.419  mm,	Y = -212.818  mm,	Z = -241.208  mm,
	W = 0.000 deg,	P = 30.000 deg,	R = 177.467 deg
};
P[109]{
   GP1:
	UF : 0, UT : 1,		CONFIG : 'N U T, 0, 0, 0',
	X = 1213.461  mm,	Y = -210.818  mm,	Z = -241.197  mm,
	W = 0.000 deg,	P = 30.000 deg,	R = 169.103 deg
};
P[110]{
   GP1:
	UF : 0, UT : 1,		CONFIG : 'N U T, 0, 0, 0',
	X = 1213.502  mm,	Y = -208.818  mm,	Z = -241.185  mm,
	W = 0.000 deg,	P = 30.000 deg,	R = 160.740 deg
};
P[111]{
   GP1:
	UF : 0, UT : 1,		CONFIG : 'N U T, 0, 0, 0',
	X = 1213.544  mm,	Y = -206.819  mm,	Z = -241.173  mm,
	W = 0.000 deg,	P = 30.000 deg,	R = 152.376 deg
};
P[112]{
   GP1:
	UF : 0, UT : 1,		CONFIG : 'N U T, 0, 0, 0',
	X = 1213.586  mm,	Y = -204.819  mm,	Z = -241.161  mm,
	W = 0.000 deg,	P = 30.000 deg,	R = 144.013 deg
};
P[113]{
   GP1:
	UF : 0, UT : 1,		CONFIG : 'N U T, 0, 0, 0',
	X = 1213.630  mm,	Y = -202.771  mm,	Z = -241.150  mm,
	W = 0.000 deg,	P = 30.000 deg,	R = 136.993 deg
};
P[114]{
   GP1:
	UF : 0, UT : 1,		CONFIG : 'N U T, 0, 0, 0',
	X = 1222.330  mm,	Y = -206.354  mm,	Z = -241.160  mm,
	W = 0.000 deg,	P = 30.000 deg,	R = 136.993 deg
};
P[115]{
   GP1:
	UF : 0, UT : 1,		CONFIG : 'N U T, 0, 0, 0',
	X = 1216.370  mm,	Y = -198.083  mm,	Z = -241.419  mm,
	W = 0.000 deg,	P = 30.000 deg,	R = 136.993 deg
};
P[116]{
   GP1:
	UF : 0, UT : 1,		CONFIG : 'N U T, 0, 0, 0',
	X = 1217.723  mm,	Y = -196.633  mm,	Z = -241.678  mm,
	W = 0.000 deg,	P = 30.000 deg,	R = 136.993 deg
};
P[117]{
   GP1:
	UF : 0, UT : 1,		CONFIG : 'N U T, 0, 0, 0',
	X = 1219.076  mm,	Y = -195.183  mm,	Z = -241.937  mm,
	W = 0.000 deg,	P = 30.000 deg,	R = 136.993 deg
};
P[118]{
   GP1:
	UF : 0, UT : 1,		CONFIG : 'N U T, 0, 0, 0',
	X = 1220.429  mm,	Y = -193.733  mm,	Z = -242.196  mm,
	W = 0.000 deg,	P = 30.000 deg,	R = 136.993 deg
};
P[119]{
   GP1:
	UF : 0, UT : 1,		CONFIG : 'N U T, 0, 0, 0',
	X = 1221.781  mm,	Y = -192.282  mm,	Z = -242.455  mm,
	W = 0.000 deg,	P = 30.000 deg,	R = 136.993 deg
};
P[120]{
   GP1:
	UF : 0, UT : 1,		CONFIG : 'N U T, 0, 0, 0',
	X = 1223.134  mm,	Y = -190.832  mm,	Z = -242.714  mm,
	W = 0.000 deg,	P = 30.000 deg,	R = 136.993 deg
};
P[121]{
   GP1:
	UF : 0, UT : 1,		CONFIG : 'N U T, 0, 0, 0',
	X = 1224.487  mm,	Y = -189.382  mm,	Z = -242.973  mm,
	W = 0.000 deg,	P = 30.000 deg,	R = 136.993 deg
};
P[122]{
   GP1:
	UF : 0, UT : 1,		CONFIG : 'N U T, 0, 0, 0',
	X = 1233.152  mm,	Y = -194.753  mm,	Z = -243.232  mm,
	W = 0.000 deg,	P = 30.000 deg,	R = 136.993 deg
};
P[123]{
   GP1:
	UF : 0, UT : 1,		CONFIG : 'N U T, 0, 0, 0',
	X = 1234.505  mm,	Y = -193.302  mm,	Z = -243.491  mm,
	W = 0.000 deg,	P = 30.000 deg,	R = 136.993 deg
};
P[124]{
   GP1:
	UF : 0, UT : 1,		CONFIG : 'N U T, 0, 0, 0',
	X = 1228.545  mm,	Y = -185.031  mm,	Z = -243.750  mm,
	W = 0.000 deg,	P = 30.000 deg,	R = 136.993 deg
};
P[125]{
   GP1:
	UF : 0, UT : 1,		CONFIG : 'N U T, 0, 0, 0',
	X = 1229.897  mm,	Y = -183.581  mm,	Z = -244.009  mm,
	W = 0.000 deg,	P = 30.000 deg,	R = 136.993 deg
};
P[126]{
   GP1:
	UF : 0, UT : 1,		CONFIG : 'N U T, 0, 0, 0',
	X = 1231.250  mm,	Y = -182.131  mm,	Z = -244.268  mm,
	W = 0.000 deg,	P = 30.000 deg,	R = 136.993 deg
};
P[127]{
   GP1:
	UF : 0, UT : 1,		CONFIG : 'N U T, 0, 0, 0',
	X = 1232.603  mm,	Y = -180.681  mm,	Z = -244.527  mm,
	W = 0.000 deg,	P = 30.000 deg,	R = 136.993 deg
};
P[128]{
   GP1:
	UF : 0, UT : 1,		CONFIG : 'N U T, 0, 0, 0',
	X = 1233.955  mm,	Y = -179.230  mm,	Z = -244.786  mm,
	W = 0.000 deg,	P = 30.000 deg,	R = 136.993 deg
};
P[129]{
   GP1:
	UF : 0, UT : 1,		CONFIG : 'N U T, 0, 0, 0',
	X = 1235.308  mm,	Y = -177.780  mm,	Z = -245.045  mm,
	W = 0.000 deg,	P = 30.000 deg,	R = 136.993 deg
};
P[130]{
   GP1:
	UF : 0, UT : 1,		CONFIG : 'N U T, 0, 0, 0',
	X = 1236.661  mm,	Y = -176.330  mm,	Z = -245.304  mm,
	W = 0.000 deg,	P = 30.000 deg,	R = 136.993 deg
};
P[131]{
   GP1:
	UF : 0, UT : 1,		CONFIG : 'N U T, 0, 0, 0',
	X = 1238.014  mm,	Y = -174.880  mm,	Z = -245.563  mm,
	W = 0.000 deg,	P = 30.000 deg,	R = 136.993 deg
};
P[132]{
   GP1:
	UF : 0, UT : 1,		CONFIG : 'N U T, 0, 0, 0',
	X = 1239.366  mm,	Y = -173.430  mm,	Z = -245.822  mm,
	W = 0.000 deg,	P = 30.000 deg,	R = 136.993 deg
};
P[133]{
   GP1:
	UF : 0, UT : 1,		CONFIG : 'N U T, 0, 0, 0',
	X = 1240.719  mm,	Y = -171.979  mm,	Z = -246.081  mm,
	W = 0.000 deg,	P = 30.000 deg,	R = 136.993 deg
};
P[134]{
   GP1:
	UF : 0, UT : 1,		CONFIG : 'N U T, 0, 0, 0',
	X = 1249.384  mm,	Y = -177.350  mm,	Z = -246.340  mm,
	W = 0.000 deg,	P = 30.000 deg,	R = 146.203 deg
};
P[135]{
   GP1:
	UF : 0, UT : 1,		CONFIG : 'N U T, 0, 0, 0',
	X = 1250.737  mm,	Y = -175.900  mm,	Z = -246.599  mm,
	W = 0.000 deg,	P = 30.000 deg,	R = 155.088 deg
};
P[136]{
   GP1:
	UF : 0, UT : 1,		CONFIG : 'N U T, 0, 0, 0',
	X = 1252.090  mm,	Y = -174.450  mm,	Z = -246.858  mm,
	W = 0.000 deg,	P = 30.000 deg,	R = 163.973 deg
};
P[137]{
   GP1:
	UF : 0, UT : 1,		CONFIG : 'N U T, 0, 0, 0',
	X = 1253.442  mm,	Y = -172.999  mm,	Z = -247.117  mm,
	W = 0.000 deg,	P = 30.000 deg,	R = 172.858 deg
};
P[138]{
   GP1:
	UF : 0, UT : 1,		CONFIG : 'N U T, 0, 0, 0',
	X = 1254.795  mm,	Y = -171.549  mm,	Z = -247.376  mm,
	W = 0.000 deg,	P = 30.000 deg,	R = -178.582 deg
};
P[139]{
   GP1:
	UF : 0, UT : 1,		CONFIG : 'N U T, 0, 0, 0',
	X = 1256.297  mm,	Y = -169.895  mm,	Z = -247.596  mm,
	W = 0.000 deg,	P = 30.000 deg,	R = -178.582 deg
};
P[140]{
   GP1:
	UF : 0, UT : 1,		CONFIG : 'N U T, 0, 0, 0',
	X = 1257.280  mm,	Y = -166.483  mm,	Z = -247.589  mm,
	W = 0.000 deg,	P = 30.000 deg,	R = -178.582 deg
};
P[141]{
   GP1:
	UF : 0, UT : 1,		CONFIG : 'N U T, 0, 0, 0',
	X = 1257.231  mm,	Y = -164.484  mm,	Z = -247.542  mm,
	W = 0.000 deg,	P = 30.000 deg,	R = -178.582 deg
};
P[142]{
   GP1:
	UF : 0, UT : 1,		CONFIG : 'N U T, 0, 0, 0',
	X = 1257.181  mm,	Y = -162.485  mm,	Z = -247.494  mm,
	W = 0.000 deg,	P = 30.000 deg,	R = -178.582 deg
};
P[143]{
   GP1:
	UF : 0, UT : 1,		CONFIG : 'N U T, 0, 0, 0',
	X = 1247.135  mm,	Y = -160.734  mm,	Z = -247.447  mm,
	W = 0.000 deg,	P = 30.000 deg,	R = -178.582 deg
};
P[144]{
   GP1:
	UF : 0, UT : 1,		CONFIG : 'N U T, 0, 0, 0',
	X = 1247.085  mm,	Y = -158.735  mm,	Z = -247.399  mm,
	W = 0.000 deg,	P = 30.000 deg,	R = -178.582 deg
};
P[145]{
   GP1:
	UF : 0, UT : 1,		CONFIG : 'N U T, 0, 0, 0',
	X = 1257.033  mm,	Y = -156.489  mm,	Z = -247.352  mm,
	W = 0.000 deg,	P = 30.000 deg,	R = -178.582 deg
};
P[146]{
   GP1:
	UF : 0, UT : 1,		CONFIG : 'N U T, 0, 0, 0',
	X = 1256.983  mm,	Y = -154.490  mm,	Z = -247.304  mm,
	W = 0.000 deg,	P = 30.000 deg,	R = -178.582 deg
};
P[147]{
   GP1:
	UF : 0, UT : 1,		CONFIG : 'N U T, 0, 0, 0',
	X = 1256.934  mm,	Y = -152.491  mm,	Z = -247.257  mm,
	W = 0.000 deg,	P = 30.000 deg,	R = -178.582 deg
};
P[148]{
   GP1:
	UF : 0, UT : 1,		CONFIG : 'N U T, 0, 0, 0',
	X = 1246.888  mm,	Y = -150.740  mm,	Z = -247.209  mm,
	W = 0.000 deg,	P = 30.000 deg,	R = -178.582 deg
};
P[149]{
   GP1:
	UF : 0, UT : 1,		CONFIG : 'N U T, 0, 0, 0',
	X = 1246.838  mm,	Y = -148.741  mm,	Z = -247.162  mm,
	W = 0.000 deg,	P = 30.000 deg,	R = -178.582 deg
};
P[150]{
   GP1:
	UF : 0, UT : 1,		CONFIG : 'N U T, 0, 0, 0',
	X = 1256.786  mm,	Y = -146.494  mm,	Z = -247.115  mm,
	W = 0.000 deg,	P = 30.000 deg,	R = -178.582 deg
};
P[151]{
   GP1:
	UF : 0, UT : 1,		CONFIG : 'N U T, 0, 0, 0',
	X = 1256.736  mm,	Y = -144.496  mm,	Z = -247.067  mm,
	W = 0.000 deg,	P = 30.000 deg,	R = -178.582 deg
};
P[152]{
   GP1:
	UF : 0, UT : 1,		CONFIG : 'N U T, 0, 0, 0',
	X = 1256.687  mm,	Y = -142.497  mm,	Z = -247.020  mm,
	W = 0.000 deg,	P = 30.000 deg,	R = -178.582 deg
};
P[153]{
   GP1:
	UF : 0, UT : 1,		CONFIG : 'N U T, 0, 0, 0',
	X = 1246.640  mm,	Y = -140.745  mm,	Z = -246.972  mm,
	W = 0.000 deg,	P = 30.000 deg,	R = -178.582 deg
};
P[154]{
   GP1:
	UF : 0, UT : 1,		CONFIG : 'N U T, 0, 0, 0',
	X = 1246.591  mm,	Y = -138.747  mm,	Z = -246.925  mm,
	W = 0.000 deg,	P = 30.000 deg,	R = -178.582 deg
};
P[155]{
   GP1:
	UF : 0, UT : 1,		CONFIG : 'N U T, 0, 0, 0',
	X = 1256.538  mm,	Y = -136.500  mm,	Z = -246.877  mm,
	W = 0.000 deg,	P = 30.000 deg,	R = -178.582 deg
};
P[156]{
   GP1:
	UF : 0, UT : 1,		CONFIG : 'N U T, 0, 0, 0',
	X = 1256.489  mm,	Y = -134.502  mm,	Z = -246.830  mm,
	W = 0.000 deg,	P = 30.000 deg,	R = -178.582 deg
};
P[157]{
   GP1:
	UF : 0, UT : 1,		CONFIG : 'N U T, 0, 0, 0',
	X = 1256.439  mm,	Y = -132.503  mm,	Z = -246.782  mm,
	W = 0.000 deg,	P = 30.000 deg,	R = -178.582 deg
};
P[158]{
   GP1:
	UF : 0, UT : 1,		CONFIG : 'N U T, 0, 0, 0',
	X = 1246.393  mm,	Y = -130.751  mm,	Z = -246.735  mm,
	W = 0.000 deg,	P = 30.000 deg,	R = -178.582 deg
};
P[159]{
   GP1:
	UF : 0, UT : 1,		CONFIG : 'N U T, 0, 0, 0',
	X = 1246.343  mm,	Y = -128.752  mm,	Z = -246.688  mm,
	W = 0.000 deg,	P = 30.000 deg,	R = -178.582 deg
};
P[160]{
   GP1:
	UF : 0, UT : 1,		CONFIG : 'N U T, 0, 0, 0',
	X = 1256.291  mm,	Y = -126.506  mm,	Z = -246.640  mm,
	W = 0.000 deg,	P = 30.000 deg,	R = -178.582 deg
};
P[161]{
   GP1:
	UF : 0, UT : 1,		CONFIG : 'N U T, 0, 0, 0',
	X = 1256.241  mm,	Y = -124.507  mm,	Z = -246.593  mm,
	W = 0.000 deg,	P = 30.000 deg,	R = -178.582 deg
};
P[162]{
   GP1:
	UF : 0, UT : 1,		CONFIG : 'N U T, 0, 0, 0',
	X = 1256.192  mm,	Y = -122.509  mm,	Z = -246.545  mm,
	W = 0.000 deg,	P = 30.000 deg,	R = -178.582 deg
};
P[163]{
   GP1:
	UF : 0, UT : 1,		CONFIG : 'N U T, 0, 0, 0',
	X = 1246.146  mm,	Y = -120.757  mm,	Z = -246.498  mm,
	W = 0.000 deg,	P = 30.000 deg,	R = -178.582 deg
};
P[164]{
   GP1:
	UF : 0, UT : 1,		CONFIG : 'N U T, 0, 0, 0',
	X = 1246.096  mm,	Y = -118.758  mm,	Z = -246.450  mm,
	W = 0.000 deg,	P = 30.000 deg,	R = -178.582 deg
};
P[165]{
   GP1:
	UF : 0, UT : 1,		CONFIG : 'N U T, 0, 0, 0',
	X = 1256.044  mm,	Y = -116.512  mm,	Z = -246.403  mm,
	W = 0.000 deg,	P = 30.000 deg,	R = -168.810 deg
};
P[166]{
   GP1:
	UF : 0, UT : 1,		CONFIG : 'N U T, 0, 0, 0',
	X = 1255.994  mm,	Y = -114.513  mm,	Z = -246.355  mm,
	W = 0.000 deg,	P = 30.000 deg,	R = -160.309 deg
};
P[167]{
   GP1:
	UF : 0, UT : 1,		CONFIG : 'N U T, 0, 0, 0',
	X = 1255.945  mm,	Y = -112.514  mm,	Z = -246.308  mm,
	W = 0.000 deg,	P = 30.000 deg,	R = -151.809 deg
};
P[168]{
   GP1:
	UF : 0, UT : 1,		CONFIG : 'N U T, 0, 0, 0',
	X = 1255.895  mm,	Y = -110.516  mm,	Z = -246.261  mm,
	W = 0.000 deg,	P = 30.000 deg,	R = -143.308 deg
};
P[169]{
   GP1:
	UF : 0, UT : 1,		CONFIG : 'N U T, 0, 0, 0',
	X = 1255.846  mm,	Y = -108.517  mm,	Z = -246.213  mm,
	W = 0.000 deg,	P = 30.000 deg,	R = -136.078 deg
};
P[170]{
   GP1:
	UF : 0, UT : 1,		CONFIG : 'N U T, 0, 0, 0',
	X = 1254.519  mm,	Y = -105.187  mm,	Z = -246.212  mm,
	W = 0.000 deg,	P = 30.000 deg,	R = -136.078 deg
};
P[171]{
   GP1:
	UF : 0, UT : 1,		CONFIG : 'N U T, 0, 0, 0',
	X = 1253.117  mm,	Y = -103.730  mm,	Z = -245.927  mm,
	W = 0.000 deg,	P = 30.000 deg,	R = -136.078 deg
};
P[172]{
   GP1:
	UF : 0, UT : 1,		CONFIG : 'N U T, 0, 0, 0',
	X = 1244.541  mm,	Y = -109.241  mm,	Z = -245.634  mm,
	W = 0.000 deg,	P = 30.000 deg,	R = -136.078 deg
};
P[173]{
   GP1:
	UF : 0, UT : 1,		CONFIG : 'N U T, 0, 0, 0',
	X = 1243.169  mm,	Y = -107.816  mm,	Z = -245.341  mm,
	W = 0.000 deg,	P = 30.000 deg,	R = -136.078 deg
};
P[174]{
   GP1:
	UF : 0, UT : 1,		CONFIG : 'N U T, 0, 0, 0',
	X = 1241.797  mm,	Y = -106.391  mm,	Z = -245.048  mm,
	W = 0.000 deg,	P = 30.000 deg,	R = -136.078 deg
};
P[175]{
   GP1:
	UF : 0, UT : 1,		CONFIG : 'N U T, 0, 0, 0',
	X = 1240.424  mm,	Y = -104.966  mm,	Z = -244.755  mm,
	W = 0.000 deg,	P = 30.000 deg,	R = -136.078 deg
};
P[176]{
   GP1:
	UF : 0, UT : 1,		CONFIG : 'N U T, 0, 0, 0',
	X = 1239.052  mm,	Y = -103.541  mm,	Z = -244.462  mm,
	W = 0.000 deg,	P = 30.000 deg,	R = -136.078 deg
};
P[177]{
   GP1:
	UF : 0, UT : 1,		CONFIG : 'N U T, 0, 0, 0',
	X = 1244.883  mm,	Y = -95.179  mm,	Z = -244.169  mm,
	W = 0.000 deg,	P = 30.000 deg,	R = -136.078 deg
};
P[178]{
   GP1:
	UF : 0, UT : 1,		CONFIG : 'N U T, 0, 0, 0',
	X = 1236.307  mm,	Y = -100.691  mm,	Z = -243.876  mm,
	W = 0.000 deg,	P = 30.000 deg,	R = -136.078 deg
};
P[179]{
   GP1:
	UF : 0, UT : 1,		CONFIG : 'N U T, 0, 0, 0',
	X = 1234.935  mm,	Y = -99.266  mm,	Z = -243.583  mm,
	W = 0.000 deg,	P = 30.000 deg,	R = -136.078 deg
};
P[180]{
   GP1:
	UF : 0, UT : 1,		CONFIG : 'N U T, 0, 0, 0',
	X = 1233.563  mm,	Y = -97.841  mm,	Z = -243.290  mm,
	W = 0.000 deg,	P = 30.000 deg,	R = -136.078 deg
};
P[181]{
   GP1:
	UF : 0, UT : 1,		CONFIG : 'N U T, 0, 0, 0',
	X = 1232.190  mm,	Y = -96.416  mm,	Z = -242.996  mm,
	W = 0.000 deg,	P = 30.000 deg,	R = -136.078 deg
};
P[182]{
   GP1:
	UF : 0, UT : 1,		CONFIG : 'N U T, 0, 0, 0',
	X = 1230.818  mm,	Y = -94.991  mm,	Z = -242.703  mm,
	W = 0.000 deg,	P = 30.000 deg,	R = -136.078 deg
};
P[183]{
   GP1:
	UF : 0, UT : 1,		CONFIG : 'N U T, 0, 0, 0',
	X = 1229.445  mm,	Y = -93.566  mm,	Z = -242.410  mm,
	W = 0.000 deg,	P = 30.000 deg,	R = -136.078 deg
};
P[184]{
   GP1:
	UF : 0, UT : 1,		CONFIG : 'N U T, 0, 0, 0',
	X = 1228.073  mm,	Y = -92.141  mm,	Z = -242.117  mm,
	W = 0.000 deg,	P = 30.000 deg,	R = -136.078 deg
};
P[185]{
   GP1:
	UF : 0, UT : 1,		CONFIG : 'N U T, 0, 0, 0',
	X = 1226.701  mm,	Y = -90.716  mm,	Z = -241.824  mm,
	W = 0.000 deg,	P = 30.000 deg,	R = -136.078 deg
};
P[186]{
   GP1:
	UF : 0, UT : 1,		CONFIG : 'N U T, 0, 0, 0',
	X = 1225.328  mm,	Y = -89.291  mm,	Z = -241.531  mm,
	W = 0.000 deg,	P = 30.000 deg,	R = -136.078 deg
};
P[187]{
   GP1:
	UF : 0, UT : 1,		CONFIG : 'N U T, 0, 0, 0',
	X = 1223.956  mm,	Y = -87.866  mm,	Z = -241.238  mm,
	W = 0.000 deg,	P = 30.000 deg,	R = -136.078 deg
};
P[188]{
   GP1:
	UF : 0, UT : 1,		CONFIG : 'N U T, 0, 0, 0',
	X = 1229.786  mm,	Y = -79.504  mm,	Z = -240.945  mm,
	W = 0.000 deg,	P = 30.000 deg,	R = -136.078 deg
};
P[189]{
   GP1:
	UF : 0, UT : 1,		CONFIG : 'N U T, 0, 0, 0',
	X = 1228.414  mm,	Y = -78.079  mm,	Z = -240.652  mm,
	W = 0.000 deg,	P = 30.000 deg,	R = -136.078 deg
};
P[190]{
   GP1:
	UF : 0, UT : 1,		CONFIG : 'N U T, 0, 0, 0',
	X = 1219.839  mm,	Y = -83.591  mm,	Z = -240.358  mm,
	W = 0.000 deg,	P = 30.000 deg,	R = -136.078 deg
};
P[191]{
   GP1:
	UF : 0, UT : 1,		CONFIG : 'N U T, 0, 0, 0',
	X = 1218.466  mm,	Y = -82.166  mm,	Z = -240.065  mm,
	W = 0.000 deg,	P = 30.000 deg,	R = -136.078 deg
};
P[192]{
   GP1:
	UF : 0, UT : 1,		CONFIG : 'N U T, 0, 0, 0',
	X = 1217.094  mm,	Y = -80.741  mm,	Z = -239.772  mm,
	W = 0.000 deg,	P = 30.000 deg,	R = -153.864 deg
};
P[193]{
   GP1:
	UF : 0, UT : 1,		CONFIG : 'N U T, 0, 0, 0',
	X = 1215.722  mm,	Y = -79.316  mm,	Z = -239.479  mm,
	W = 0.000 deg,	P = 30.000 deg,	R = -162.894 deg
};
P[194]{
   GP1:
	UF : 0, UT : 1,		CONFIG : 'N U T, 0, 0, 0',
	X = 1214.349  mm,	Y = -77.891  mm,	Z = -239.186  mm,
	W = 0.000 deg,	P = 30.000 deg,	R = -171.924 deg
};
P[195]{
   GP1:
	UF : 0, UT : 1,		CONFIG : 'N U T, 0, 0, 0',
	X = 1212.977  mm,	Y = -76.466  mm,	Z = -238.893  mm,
	W = 0.000 deg,	P = 30.000 deg,	R = 179.046 deg
};
P[196]{
   GP1:
	UF : 0, UT : 1,		CONFIG : 'N U T, 0, 0, 0',
	X = 1211.230  mm,	Y = -73.930  mm,	Z = -238.766  mm,
	W = 0.000 deg,	P = 30.000 deg,	R = 178.771 deg
};
P[197]{
   GP1:
	UF : 0, UT : 1,		CONFIG : 'N U T, 0, 0, 0',
	X = 1211.009  mm,	Y = -71.140  mm,	Z = -238.759  mm,
	W = 0.000 deg,	P = 30.000 deg,	R = 178.771 deg
};
P[198]{
   GP1:
	UF : 0, UT : 1,		CONFIG : 'N U T, 0, 0, 0',
	X = 1211.052  mm,	Y = -69.140  mm,	Z = -238.746  mm,
	W = 0.000 deg,	P = 30.000 deg,	R = 178.771 deg
};
P[199]{
   GP1:
	UF : 0, UT : 1,		CONFIG : 'N U T, 0, 0, 0',
	X = 1211.094  mm,	Y = -67.141  mm,	Z = -238.734  mm,
	W = 0.000 deg,	P = 30.000 deg,	R = 178.771 deg
};
P[200]{
   GP1:
	UF : 0, UT : 1,		CONFIG : 'N U T, 0, 0, 0',
	X = 1211.137  mm,	Y = -65.141  mm,	Z = -238.722  mm,
	W = 0.000 deg,	P = 30.000 deg,	R = 178.771 deg
};
P[201]{
   GP1:
	UF : 0, UT : 1,		CONFIG : 'N U T, 0, 0, 0',
	X = 1211.180  mm,	Y = -63.142  mm,	Z = -238.709  mm,
	W = 0.000 deg,	P = 30.000 deg,	R = 178.771 deg
};
P[202]{
   GP1:
	UF : 0, UT : 1,		CONFIG : 'N U T, 0, 0, 0',
	X = 1221.221  mm,	Y = -61.357  mm,	Z = -238.697  mm,
	W = 0.000 deg,	P = 30.000 deg,	R = 178.771 deg
};
P[203]{
   GP1:
	UF : 0, UT : 1,		CONFIG : 'N U T, 0, 0, 0',
	X = 1221.264  mm,	Y = -59.357  mm,	Z = -238.684  mm,
	W = 0.000 deg,	P = 30.000 deg,	R = 178.771 deg
};
P[204]{
   GP1:
	UF : 0, UT : 1,		CONFIG : 'N U T, 0, 0, 0',
	X = 1211.309  mm,	Y = -57.143  mm,	Z = -238.672  mm,
	W = 0.000 deg,	P = 30.000 deg,	R = 178.771 deg
};
P[205]{
   GP1:
	UF : 0, UT : 1,		CONFIG : 'N U T, 0, 0, 0',
	X = 1211.352  mm,	Y = -55.144  mm,	Z = -238.660  mm,
	W = 0.000 deg,	P = 30.000 deg,	R = 178.771 deg
};
P[206]{
   GP1:
	UF : 0, UT : 1,		CONFIG : 'N U T, 0, 0, 0',
	X = 1211.395  mm,	Y = -53.144  mm,	Z = -238.647  mm,
	W = 0.000 deg,	P = 30.000 deg,	R = 178.771 deg
};
P[207]{
   GP1:
	UF : 0, UT : 1,		CONFIG : 'N U T, 0, 0, 0',
	X = 1211.438  mm,	Y = -51.145  mm,	Z = -238.635  mm,
	W = 0.000 deg,	P = 30.000 deg,	R = 178.771 deg
};
P[208]{
   GP1:
	UF : 0, UT : 1,		CONFIG : 'N U T, 0, 0, 0',
	X = 1211.481  mm,	Y = -49.145  mm,	Z = -238.622  mm,
	W = 0.000 deg,	P = 30.000 deg,	R = 178.771 deg
};
P[209]{
   GP1:
	UF : 0, UT : 1,		CONFIG : 'N U T, 0, 0, 0',
	X = 1211.523  mm,	Y = -47.146  mm,	Z = -238.610  mm,
	W = 0.000 deg,	P = 30.000 deg,	R = 178.771 deg
};
P[210]{
   GP1:
	UF : 0, UT : 1,		CONFIG : 'N U T, 0, 0, 0',
	X = 1221.564  mm,	Y = -45.361  mm,	Z = -238.598  mm,
	W = 0.000 deg,	P = 30.000 deg,	R = 178.771 deg
};
P[211]{
   GP1:
	UF : 0, UT : 1,		CONFIG : 'N U T, 0, 0, 0',
	X = 1221.607  mm,	Y = -43.361  mm,	Z = -238.585  mm,
	W = 0.000 deg,	P = 30.000 deg,	R = 178.771 deg
};
P[212]{
   GP1:
	UF : 0, UT : 1,		CONFIG : 'N U T, 0, 0, 0',
	X = 1211.652  mm,	Y = -41.147  mm,	Z = -238.573  mm,
	W = 0.000 deg,	P = 30.000 deg,	R = 178.771 deg
};
P[213]{
   GP1:
	UF : 0, UT : 1,		CONFIG : 'N U T, 0, 0, 0',
	X = 1211.695  mm,	Y = -39.148  mm,	Z = -238.560  mm,
	W = 0.000 deg,	P = 30.000 deg,	R = 178.771 deg
};
P[214]{
   GP1:
	UF : 0, UT : 1,		CONFIG : 'N U T, 0, 0, 0',
	X = 1211.738  mm,	Y = -37.148  mm,	Z = -238.548  mm,
	W = 0.000 deg,	P = 30.000 deg,	R = 178.771 deg
};
P[215]{
   GP1:
	UF : 0, UT : 1,		CONFIG : 'N U T, 0, 0, 0',
	X = 1211.781  mm,	Y = -35.149  mm,	Z = -238.536  mm,
	W = 0.000 deg,	P = 30.000 deg,	R = 178.771 deg
};
P[216]{
   GP1:
	UF : 0, UT : 1,		CONFIG : 'N U T, 0, 0, 0',
	X = 1211.824  mm,	Y = -33.149  mm,	Z = -238.523  mm,
	W = 0.000 deg,	P = 30.000 deg,	R = 178.771 deg
};
P[217]{
   GP1:
	UF : 0, UT : 1,		CONFIG : 'N U T, 0, 0, 0',
	X = 1211.867  mm,	Y = -31.150  mm,	Z = -238.511  mm,
	W = 0.000 deg,	P = 30.000 deg,	R = 178.771 deg
};
P[218]{
   GP1:
	UF : 0, UT : 1,		CONFIG : 'N U T, 0, 0, 0',
	X = 1221.907  mm,	Y = -29.365  mm,	Z = -238.498  mm,
	W = 0.000 deg,	P = 30.000 deg,	R = 178.771 deg
};
P[219]{
   GP1:
	UF : 0, UT : 1,		CONFIG : 'N U T, 0, 0, 0',
	X = 1221.950  mm,	Y = -27.365  mm,	Z = -238.486  mm,
	W = 0.000 deg,	P = 30.000 deg,	R = 178.771 deg
};
P[220]{
   GP1:
	UF : 0, UT : 1,		CONFIG : 'N U T, 0, 0, 0',
	X = 1211.995  mm,	Y = -25.151  mm,	Z = -238.474  mm,
	W = 0.000 deg,	P = 30.000 deg,	R = 178.771 deg
};
P[221]{
   GP1:
	UF : 0, UT : 1,		CONFIG : 'N U T, 0, 0, 0',
	X = 1212.038  mm,	Y = -23.152  mm,	Z = -238.461  mm,
	W = 0.000 deg,	P = 30.000 deg,	R = 178.771 deg
};
P[222]{
   GP1:
	UF : 0, UT : 1,		CONFIG : 'N U T, 0, 0, 0',
	X = 1212.081  mm,	Y = -21.152  mm,	Z = -238.449  mm,
	W = 0.000 deg,	P = 30.000 deg,	R = 165.090 deg
};
P[223]{
   GP1:
	UF : 0, UT : 1,		CONFIG : 'N U T, 0, 0, 0',
	X = 1212.124  mm,	Y = -19.153  mm,	Z = -238.436  mm,
	W = 0.000 deg,	P = 30.000 deg,	R = 156.355 deg
};
P[224]{
   GP1:
	UF : 0, UT : 1,		CONFIG : 'N U T, 0, 0, 0',
	X = 1212.167  mm,	Y = -17.153  mm,	Z = -238.424  mm,
	W = 0.000 deg,	P = 30.000 deg,	R = 147.620 deg
};
P[225]{
   GP1:
	UF : 0, UT : 1,		CONFIG : 'N U T, 0, 0, 0',
	X = 1212.210  mm,	Y = -15.154  mm,	Z = -238.412  mm,
	W = 0.000 deg,	P = 30.000 deg,	R = 138.885 deg
};
P[226]{
   GP1:
	UF : 0, UT : 1,		CONFIG : 'N U T, 0, 0, 0',
	X = 1212.254  mm,	Y = -13.126  mm,	Z = -238.399  mm,
	W = 0.000 deg,	P = 30.000 deg,	R = 135.096 deg
};
P[227]{
   GP1:
	UF : 0, UT : 1,		CONFIG : 'N U T, 0, 0, 0',
	X = 1220.820  mm,	Y = -16.803  mm,	Z = -238.405  mm,
	W = 0.000 deg,	P = 30.000 deg,	R = 135.096 deg
};
P[228]{
   GP1:
	UF : 0, UT : 1,		CONFIG : 'N U T, 0, 0, 0',
	X = 1215.136  mm,	Y = -8.341  mm,	Z = -238.679  mm,
	W = 0.000 deg,	P = 30.000 deg,	R = 135.096 deg
};
P[229]{
   GP1:
	UF : 0, UT : 1,		CONFIG : 'N U T, 0, 0, 0',
	X = 1216.534  mm,	Y = -6.937  mm,	Z = -238.954  mm,
	W = 0.000 deg,	P = 30.000 deg,	R = 135.096 deg
};
P[230]{
   GP1:
	UF : 0, UT : 1,		CONFIG : 'N U T, 0, 0, 0',
	X = 1225.015  mm,	Y = -12.593  mm,	Z = -239.228  mm,
	W = 0.000 deg,	P = 30.000 deg,	R = 135.096 deg
};
P[231]{
   GP1:
	UF : 0, UT : 1,		CONFIG : 'N U T, 0, 0, 0',
	X = 1226.414  mm,	Y = -11.190  mm,	Z = -239.503  mm,
	W = 0.000 deg,	P = 30.000 deg,	R = 135.096 deg
};
P[232]{
   GP1:
	UF : 0, UT : 1,		CONFIG : 'N U T, 0, 0, 0',
	X = 1220.730  mm,	Y = -2.728  mm,	Z = -239.777  mm,
	W = 0.000 deg,	P = 30.000 deg,	R = 135.096 deg
};
P[233]{
   GP1:
	UF : 0, UT : 1,		CONFIG : 'N U T, 0, 0, 0',
	X = 1222.128  mm,	Y = -1.325  mm,	Z = -240.052  mm,
	W = 0.000 deg,	P = 30.000 deg,	R = 135.096 deg
};
P[234]{
   GP1:
	UF : 0, UT : 1,		CONFIG : 'N U T, 0, 0, 0',
	X = 1230.609  mm,	Y = -6.981  mm,	Z = -240.326  mm,
	W = 0.000 deg,	P = 30.000 deg,	R = 135.096 deg
};
P[235]{
   GP1:
	UF : 0, UT : 1,		CONFIG : 'N U T, 0, 0, 0',
	X = 1232.008  mm,	Y = -5.578  mm,	Z = -240.601  mm,
	W = 0.000 deg,	P = 30.000 deg,	R = 135.096 deg
};
P[236]{
   GP1:
	UF : 0, UT : 1,		CONFIG : 'N U T, 0, 0, 0',
	X = 1226.323  mm,	Y = 2.885  mm,	Z = -240.875  mm,
	W = 0.000 deg,	P = 30.000 deg,	R = 135.096 deg
};
P[237]{
   GP1:
	UF : 0, UT : 1,		CONFIG : 'N U T, 0, 0, 0',
	X = 1227.722  mm,	Y = 4.288  mm,	Z = -241.150  mm,
	W = 0.000 deg,	P = 30.000 deg,	R = 135.096 deg
};
P[238]{
   GP1:
	UF : 0, UT : 1,		CONFIG : 'N U T, 0, 0, 0',
	X = 1236.203  mm,	Y = -1.368  mm,	Z = -241.424  mm,
	W = 0.000 deg,	P = 30.000 deg,	R = 135.096 deg
};
P[239]{
   GP1:
	UF : 0, UT : 1,		CONFIG : 'N U T, 0, 0, 0',
	X = 1237.602  mm,	Y = 0.035  mm,	Z = -241.699  mm,
	W = 0.000 deg,	P = 30.000 deg,	R = 135.096 deg
};
P[240]{
   GP1:
	UF : 0, UT : 1,		CONFIG : 'N U T, 0, 0, 0',
	X = 1231.917  mm,	Y = 8.498  mm,	Z = -241.973  mm,
	W = 0.000 deg,	P = 30.000 deg,	R = 135.096 deg
};
P[241]{
   GP1:
	UF : 0, UT : 1,		CONFIG : 'N U T, 0, 0, 0',
	X = 1233.316  mm,	Y = 9.901  mm,	Z = -242.247  mm,
	W = 0.000 deg,	P = 30.000 deg,	R = 135.096 deg
};
P[242]{
   GP1:
	UF : 0, UT : 1,		CONFIG : 'N U T, 0, 0, 0',
	X = 1241.797  mm,	Y = 4.245  mm,	Z = -242.522  mm,
	W = 0.000 deg,	P = 30.000 deg,	R = 135.096 deg
};
P[243]{
   GP1:
	UF : 0, UT : 1,		CONFIG : 'N U T, 0, 0, 0',
	X = 1243.196  mm,	Y = 5.648  mm,	Z = -242.796  mm,
	W = 0.000 deg,	P = 30.000 deg,	R = 135.096 deg
};
P[244]{
   GP1:
	UF : 0, UT : 1,		CONFIG : 'N U T, 0, 0, 0',
	X = 1237.511  mm,	Y = 14.110  mm,	Z = -243.071  mm,
	W = 0.000 deg,	P = 30.000 deg,	R = 135.096 deg
};
P[245]{
   GP1:
	UF : 0, UT : 1,		CONFIG : 'N U T, 0, 0, 0',
	X = 1238.910  mm,	Y = 15.513  mm,	Z = -243.345  mm,
	W = 0.000 deg,	P = 30.000 deg,	R = 135.096 deg
};
P[246]{
   GP1:
	UF : 0, UT : 1,		CONFIG : 'N U T, 0, 0, 0',
	X = 1247.391  mm,	Y = 9.857  mm,	Z = -243.620  mm,
	W = 0.000 deg,	P = 30.000 deg,	R = 135.096 deg
};
P[247]{
   GP1:
	UF : 0, UT : 1,		CONFIG : 'N U T, 0, 0, 0',
	X = 1248.790  mm,	Y = 11.261  mm,	Z = -243.894  mm,
	W = 0.000 deg,	P = 30.000 deg,	R = 144.470 deg
};
P[248]{
   GP1:
	UF : 0, UT : 1,		CONFIG : 'N U T, 0, 0, 0',
	X = 1250.188  mm,	Y = 12.664  mm,	Z = -244.169  mm,
	W = 0.000 deg,	P = 30.000 deg,	R = 153.662 deg
};
P[249]{
   GP1:
	UF : 0, UT : 1,		CONFIG : 'N U T, 0, 0, 0',
	X = 1251.587  mm,	Y = 14.067  mm,	Z = -244.443  mm,
	W = 0.000 deg,	P = 30.000 deg,	R = 162.855 deg
};
P[250]{
   GP1:
	UF : 0, UT : 1,		CONFIG : 'N U T, 0, 0, 0',
	X = 1252.985  mm,	Y = 15.470  mm,	Z = -244.718  mm,
	W = 0.000 deg,	P = 30.000 deg,	R = 172.047 deg
};
P[251]{
   GP1:
	UF : 0, UT : 1,		CONFIG : 'N U T, 0, 0, 0',
	X = 1254.384  mm,	Y = 16.873  mm,	Z = -244.992  mm,
	W = 0.000 deg,	P = 30.000 deg,	R = -178.943 deg
};
P[252]{
   GP1:
	UF : 0, UT : 1,		CONFIG : 'N U T, 0, 0, 0',
	X = 1256.030  mm,	Y = 18.639  mm,	Z = -245.203  mm,
	W = 0.000 deg,	P = 30.000 deg,	R = -178.943 deg
};
P[253]{
   GP1:
	UF : 0, UT : 1,		CONFIG : 'N U T, 0, 0, 0',
	X = 1246.907  mm,	Y = 21.853  mm,	Z = -245.196  mm,
	W = 0.000 deg,	P = 30.000 deg,	R = -178.943 deg
};
P[254]{
   GP1:
	UF : 0, UT : 1,		CONFIG : 'N U T, 0, 0, 0',
	X = 1246.870  mm,	Y = 23.852  mm,	Z = -245.166  mm,
	W = 0.000 deg,	P = 30.000 deg,	R = -178.943 deg
};
P[255]{
   GP1:
	UF : 0, UT : 1,		CONFIG : 'N U T, 0, 0, 0',
	X = 1246.833  mm,	Y = 25.852  mm,	Z = -245.137  mm,
	W = 0.000 deg,	P = 30.000 deg,	R = -178.943 deg
};
P[256]{
   GP1:
	UF : 0, UT : 1,		CONFIG : 'N U T, 0, 0, 0',
	X = 1246.797  mm,	Y = 27.851  mm,	Z = -245.107  mm,
	W = 0.000 deg,	P = 30.000 deg,	R = -178.943 deg
};
P[257]{
   GP1:
	UF : 0, UT : 1,		CONFIG : 'N U T, 0, 0, 0',
	X = 1246.760  mm,	Y = 29.850  mm,	Z = -245.078  mm,
	W = 0.000 deg,	P = 30.000 deg,	R = -178.943 deg
};
P[258]{
   GP1:
	UF : 0, UT : 1,		CONFIG : 'N U T, 0, 0, 0',
	X = 1246.723  mm,	Y = 31.850  mm,	Z = -245.048  mm,
	W = 0.000 deg,	P = 30.000 deg,	R = -178.943 deg
};
P[259]{
   GP1:
	UF : 0, UT : 1,		CONFIG : 'N U T, 0, 0, 0',
	X = 1256.684  mm,	Y = 34.034  mm,	Z = -245.019  mm,
	W = 0.000 deg,	P = 30.000 deg,	R = -178.943 deg
};
P[260]{
   GP1:
	UF : 0, UT : 1,		CONFIG : 'N U T, 0, 0, 0',
	X = 1256.647  mm,	Y = 36.033  mm,	Z = -244.989  mm,
	W = 0.000 deg,	P = 30.000 deg,	R = -178.943 deg
};
P[261]{
   GP1:
	UF : 0, UT : 1,		CONFIG : 'N U T, 0, 0, 0',
	X = 1246.612  mm,	Y = 37.848  mm,	Z = -244.960  mm,
	W = 0.000 deg,	P = 30.000 deg,	R = -178.943 deg
};
P[262]{
   GP1:
	UF : 0, UT : 1,		CONFIG : 'N U T, 0, 0, 0',
	X = 1246.575  mm,	Y = 39.848  mm,	Z = -244.930  mm,
	W = 0.000 deg,	P = 30.000 deg,	R = -178.943 deg
};
P[263]{
   GP1:
	UF : 0, UT : 1,		CONFIG : 'N U T, 0, 0, 0',
	X = 1246.538  mm,	Y = 41.847  mm,	Z = -244.901  mm,
	W = 0.000 deg,	P = 30.000 deg,	R = -178.943 deg
};
P[264]{
   GP1:
	UF : 0, UT : 1,		CONFIG : 'N U T, 0, 0, 0',
	X = 1246.501  mm,	Y = 43.847  mm,	Z = -244.871  mm,
	W = 0.000 deg,	P = 30.000 deg,	R = -178.943 deg
};
P[265]{
   GP1:
	UF : 0, UT : 1,		CONFIG : 'N U T, 0, 0, 0',
	X = 1246.464  mm,	Y = 45.846  mm,	Z = -244.842  mm,
	W = 0.000 deg,	P = 30.000 deg,	R = -178.943 deg
};
P[266]{
   GP1:
	UF : 0, UT : 1,		CONFIG : 'N U T, 0, 0, 0',
	X = 1246.427  mm,	Y = 47.845  mm,	Z = -244.812  mm,
	W = 0.000 deg,	P = 30.000 deg,	R = -178.943 deg
};
P[267]{
   GP1:
	UF : 0, UT : 1,		CONFIG : 'N U T, 0, 0, 0',
	X = 1246.391  mm,	Y = 49.845  mm,	Z = -244.782  mm,
	W = 0.000 deg,	P = 30.000 deg,	R = -178.943 deg
};
P[268]{
   GP1:
	UF : 0, UT : 1,		CONFIG : 'N U T, 0, 0, 0',
	X = 1246.354  mm,	Y = 51.844  mm,	Z = -244.753  mm,
	W = 0.000 deg,	P = 30.000 deg,	R = -178.943 deg
};
P[269]{
   GP1:
	UF : 0, UT : 1,		CONFIG : 'N U T, 0, 0, 0',
	X = 1246.317  mm,	Y = 53.844  mm,	Z = -244.723  mm,
	W = 0.000 deg,	P = 30.000 deg,	R = -178.943 deg
};
P[270]{
   GP1:
	UF : 0, UT : 1,		CONFIG : 'N U T, 0, 0, 0',
	X = 1256.278  mm,	Y = 56.028  mm,	Z = -244.694  mm,
	W = 0.000 deg,	P = 30.000 deg,	R = -178.943 deg
};
P[271]{
   GP1:
	UF : 0, UT : 1,		CONFIG : 'N U T, 0, 0, 0',
	X = 1256.241  mm,	Y = 58.027  mm,	Z = -244.664  mm,
	W = 0.000 deg,	P = 30.000 deg,	R = -178.943 deg
};
P[272]{
   GP1:
	UF : 0, UT : 1,		CONFIG : 'N U T, 0, 0, 0',
	X = 1246.206  mm,	Y = 59.842  mm,	Z = -244.635  mm,
	W = 0.000 deg,	P = 30.000 deg,	R = -178.943 deg
};
P[273]{
   GP1:
	UF : 0, UT : 1,		CONFIG : 'N U T, 0, 0, 0',
	X = 1246.169  mm,	Y = 61.842  mm,	Z = -244.605  mm,
	W = 0.000 deg,	P = 30.000 deg,	R = -178.943 deg
};
P[274]{
   GP1:
	UF : 0, UT : 1,		CONFIG : 'N U T, 0, 0, 0',
	X = 1246.132  mm,	Y = 63.841  mm,	Z = -244.576  mm,
	W = 0.000 deg,	P = 30.000 deg,	R = -178.943 deg
};
P[275]{
   GP1:
	UF : 0, UT : 1,		CONFIG : 'N U T, 0, 0, 0',
	X = 1246.095  mm,	Y = 65.840  mm,	Z = -244.546  mm,
	W = 0.000 deg,	P = 30.000 deg,	R = -178.943 deg
};
P[276]{
   GP1:
	UF : 0, UT : 1,		CONFIG : 'N U T, 0, 0, 0',
	X = 1246.058  mm,	Y = 67.840  mm,	Z = -244.517  mm,
	W = 0.000 deg,	P = 30.000 deg,	R = -178.943 deg
};
P[277]{
   GP1:
	UF : 0, UT : 1,		CONFIG : 'N U T, 0, 0, 0',
	X = 1256.020  mm,	Y = 70.024  mm,	Z = -244.487  mm,
	W = 0.000 deg,	P = 30.000 deg,	R = -176.972 deg
};
P[278]{
   GP1:
	UF : 0, UT : 1,		CONFIG : 'N U T, 0, 0, 0',
	X = 1255.983  mm,	Y = 72.023  mm,	Z = -244.458  mm,
	W = 0.000 deg,	P = 30.000 deg,	R = -168.512 deg
};
P[279]{
   GP1:
	UF : 0, UT : 1,		CONFIG : 'N U T, 0, 0, 0',
	X = 1255.946  mm,	Y = 74.023  mm,	Z = -244.428  mm,
	W = 0.000 deg,	P = 30.000 deg,	R = -160.053 deg
};
P[280]{
   GP1:
	UF : 0, UT : 1,		CONFIG : 'N U T, 0, 0, 0',
	X = 1255.909  mm,	Y = 76.022  mm,	Z = -244.399  mm,
	W = 0.000 deg,	P = 30.000 deg,	R = -151.593 deg
};
P[281]{
   GP1:
	UF : 0, UT : 1,		CONFIG : 'N U T, 0, 0, 0',
	X = 1255.872  mm,	Y = 78.022  mm,	Z = -244.369  mm,
	W = 0.000 deg,	P = 30.000 deg,	R = -143.133 deg
};
P[282]{
   GP1:
	UF : 0, UT : 1,		CONFIG : 'N U T, 0, 0, 0',
	X = 1255.779  mm,	Y = 80.322  mm,	Z = -244.346  mm,
	W = 0.000 deg,	P = 30.000 deg,	R = -136.644 deg
};
P[283]{
   GP1:
	UF : 0, UT : 1,		CONFIG : 'N U T, 0, 0, 0',
	X = 1254.203  mm,	Y = 83.248  mm,	Z = -244.288  mm,
	W = 0.000 deg,	P = 30.000 deg,	R = -136.644 deg
};
P[284]{
   GP1:
	UF : 0, UT : 1,		CONFIG : 'N U T, 0, 0, 0',
	X = 1252.844  mm,	Y = 84.687  mm,	Z = -244.005  mm,
	W = 0.000 deg,	P = 30.000 deg,	R = -136.644 deg
};
P[285]{
   GP1:
	UF : 0, UT : 1,		CONFIG : 'N U T, 0, 0, 0',
	X = 1244.214  mm,	Y = 79.261  mm,	Z = -243.721  mm,
	W = 0.000 deg,	P = 30.000 deg,	R = -136.644 deg
};
P[286]{
   GP1:
	UF : 0, UT : 1,		CONFIG : 'N U T, 0, 0, 0',
	X = 1242.854  mm,	Y = 80.701  mm,	Z = -243.438  mm,
	W = 0.000 deg,	P = 30.000 deg,	R = -136.644 deg
};
P[287]{
   GP1:
	UF : 0, UT : 1,		CONFIG : 'N U T, 0, 0, 0',
	X = 1248.766  mm,	Y = 89.006  mm,	Z = -243.155  mm,
	W = 0.000 deg,	P = 30.000 deg,	R = -136.644 deg
};
P[288]{
   GP1:
	UF : 0, UT : 1,		CONFIG : 'N U T, 0, 0, 0',
	X = 1247.407  mm,	Y = 90.445  mm,	Z = -242.871  mm,
	W = 0.000 deg,	P = 30.000 deg,	R = -136.644 deg
};
P[289]{
   GP1:
	UF : 0, UT : 1,		CONFIG : 'N U T, 0, 0, 0',
	X = 1238.777  mm,	Y = 85.020  mm,	Z = -242.588  mm,
	W = 0.000 deg,	P = 30.000 deg,	R = -136.644 deg
};
P[290]{
   GP1:
	UF : 0, UT : 1,		CONFIG : 'N U T, 0, 0, 0',
	X = 1237.418  mm,	Y = 86.459  mm,	Z = -242.305  mm,
	W = 0.000 deg,	P = 30.000 deg,	R = -136.644 deg
};
P[291]{
   GP1:
	UF : 0, UT : 1,		CONFIG : 'N U T, 0, 0, 0',
	X = 1243.329  mm,	Y = 94.764  mm,	Z = -242.021  mm,
	W = 0.000 deg,	P = 30.000 deg,	R = -136.644 deg
};
P[292]{
   GP1:
	UF : 0, UT : 1,		CONFIG : 'N U T, 0, 0, 0',
	X = 1234.699  mm,	Y = 89.338  mm,	Z = -241.738  mm,
	W = 0.000 deg,	P = 30.000 deg,	R = -136.644 deg
};
P[293]{
   GP1:
	UF : 0, UT : 1,		CONFIG : 'N U T, 0, 0, 0',
	X = 1233.340  mm,	Y = 90.778  mm,	Z = -241.455  mm,
	W = 0.000 deg,	P = 30.000 deg,	R = -136.644 deg
};
P[294]{
   GP1:
	UF : 0, UT : 1,		CONFIG : 'N U T, 0, 0, 0',
	X = 1231.981  mm,	Y = 92.217  mm,	Z = -241.171  mm,
	W = 0.000 deg,	P = 30.000 deg,	R = -136.644 deg
};
P[295]{
   GP1:
	UF : 0, UT : 1,		CONFIG : 'N U T, 0, 0, 0',
	X = 1237.893  mm,	Y = 100.522  mm,	Z = -240.888  mm,
	W = 0.000 deg,	P = 30.000 deg,	R = -136.644 deg
};
P[296]{
   GP1:
	UF : 0, UT : 1,		CONFIG : 'N U T, 0, 0, 0',
	X = 1229.262  mm,	Y = 95.096  mm,	Z = -240.605  mm,
	W = 0.000 deg,	P = 30.000 deg,	R = -136.644 deg
};
P[297]{
   GP1:
	UF : 0, UT : 1,		CONFIG : 'N U T, 0, 0, 0',
	X = 1227.903  mm,	Y = 96.536  mm,	Z = -240.321  mm,
	W = 0.000 deg,	P = 30.000 deg,	R = -136.644 deg
};
P[298]{
   GP1:
	UF : 0, UT : 1,		CONFIG : 'N U T, 0, 0, 0',
	X = 1233.815  mm,	Y = 104.841  mm,	Z = -240.038  mm,
	W = 0.000 deg,	P = 30.000 deg,	R = -136.644 deg
};
P[299]{
   GP1:
	UF : 0, UT : 1,		CONFIG : 'N U T, 0, 0, 0',
	X = 1225.185  mm,	Y = 99.415  mm,	Z = -239.755  mm,
	W = 0.000 deg,	P = 30.000 deg,	R = -136.644 deg
};
P[300]{
   GP1:
	UF : 0, UT : 1,		CONFIG : 'N U T, 0, 0, 0',
	X = 1223.825  mm,	Y = 100.854  mm,	Z = -239.471  mm,
	W = 0.000 deg,	P = 30.000 deg,	R = -136.644 deg
};
P[301]{
   GP1:
	UF : 0, UT : 1,		CONFIG : 'N U T, 0, 0, 0',
	X = 1229.737  mm,	Y = 109.159  mm,	Z = -239.188  mm,
	W = 0.000 deg,	P = 30.000 deg,	R = -136.644 deg
};
P[302]{
   GP1:
	UF : 0, UT : 1,		CONFIG : 'N U T, 0, 0, 0',
	X = 1221.107  mm,	Y = 103.734  mm,	Z = -238.905  mm,
	W = 0.000 deg,	P = 30.000 deg,	R = -136.644 deg
};
P[303]{
   GP1:
	UF : 0, UT : 1,		CONFIG : 'N U T, 0, 0, 0',
	X = 1219.748  mm,	Y = 105.173  mm,	Z = -238.621  mm,
	W = 0.000 deg,	P = 30.000 deg,	R = -136.644 deg
};
P[304]{
   GP1:
	UF : 0, UT : 1,		CONFIG : 'N U T, 0, 0, 0',
	X = 1218.389  mm,	Y = 106.613  mm,	Z = -238.338  mm,
	W = 0.000 deg,	P = 30.000 deg,	R = -138.469 deg
};
P[305]{
   GP1:
	UF : 0, UT : 1,		CONFIG : 'N U T, 0, 0, 0',
	X = 1217.029  mm,	Y = 108.052  mm,	Z = -238.055  mm,
	W = 0.000 deg,	P = 30.000 deg,	R = -147.457 deg
};
P[306]{
   GP1:
	UF : 0, UT : 1,		CONFIG : 'N U T, 0, 0, 0',
	X = 1215.670  mm,	Y = 109.492  mm,	Z = -237.771  mm,
	W = 0.000 deg,	P = 30.000 deg,	R = -156.445 deg
};
P[307]{
   GP1:
	UF : 0, UT : 1,		CONFIG : 'N U T, 0, 0, 0',
	X = 1214.311  mm,	Y = 110.931  mm,	Z = -237.488  mm,
	W = 0.000 deg,	P = 30.000 deg,	R = -165.432 deg
};
P[308]{
   GP1:
	UF : 0, UT : 1,		CONFIG : 'N U T, 0, 0, 0',
	X = 1212.952  mm,	Y = 112.371  mm,	Z = -237.205  mm,
	W = 0.000 deg,	P = 30.000 deg,	R = -174.420 deg
};
P[309]{
   GP1:
	UF : 0, UT : 1,		CONFIG : 'N U T, 0, 0, 0',
	X = 1211.416  mm,	Y = 114.059  mm,	Z = -236.970  mm,
	W = 0.000 deg,	P = 30.000 deg,	R = 178.417 deg
};
P[310]{
   GP1:
	UF : 0, UT : 1,		CONFIG : 'N U T, 0, 0, 0',
	X = 1210.475  mm,	Y = 117.478  mm,	Z = -236.967  mm,
	W = 0.000 deg,	P = 30.000 deg,	R = 178.417 deg
};
P[311]{
   GP1:
	UF : 0, UT : 1,		CONFIG : 'N U T, 0, 0, 0',
	X = 1210.531  mm,	Y = 119.477  mm,	Z = -236.945  mm,
	W = 0.000 deg,	P = 30.000 deg,	R = 178.417 deg
};
P[312]{
   GP1:
	UF : 0, UT : 1,		CONFIG : 'N U T, 0, 0, 0',
	X = 1220.582  mm,	Y = 121.200  mm,	Z = -236.923  mm,
	W = 0.000 deg,	P = 30.000 deg,	R = 178.417 deg
};
P[313]{
   GP1:
	UF : 0, UT : 1,		CONFIG : 'N U T, 0, 0, 0',
	X = 1220.637  mm,	Y = 123.199  mm,	Z = -236.901  mm,
	W = 0.000 deg,	P = 30.000 deg,	R = 178.417 deg
};
P[314]{
   GP1:
	UF : 0, UT : 1,		CONFIG : 'N U T, 0, 0, 0',
	X = 1220.693  mm,	Y = 125.198  mm,	Z = -236.879  mm,
	W = 0.000 deg,	P = 30.000 deg,	R = 178.417 deg
};
P[315]{
   GP1:
	UF : 0, UT : 1,		CONFIG : 'N U T, 0, 0, 0',
	X = 1220.748  mm,	Y = 127.197  mm,	Z = -236.856  mm,
	W = 0.000 deg,	P = 30.000 deg,	R = 178.417 deg
};
P[316]{
   GP1:
	UF : 0, UT : 1,		CONFIG : 'N U T, 0, 0, 0',
	X = 1210.807  mm,	Y = 129.473  mm,	Z = -236.834  mm,
	W = 0.000 deg,	P = 30.000 deg,	R = 178.417 deg
};
P[317]{
   GP1:
	UF : 0, UT : 1,		CONFIG : 'N U T, 0, 0, 0',
	X = 1210.862  mm,	Y = 131.472  mm,	Z = -236.812  mm,
	W = 0.000 deg,	P = 30.000 deg,	R = 178.417 deg
};
P[318]{
   GP1:
	UF : 0, UT : 1,		CONFIG : 'N U T, 0, 0, 0',
	X = 1220.914  mm,	Y = 133.195  mm,	Z = -236.790  mm,
	W = 0.000 deg,	P = 30.000 deg,	R = 178.417 deg
};
P[319]{
   GP1:
	UF : 0, UT : 1,		CONFIG : 'N U T, 0, 0, 0',
	X = 1220.969  mm,	Y = 135.194  mm,	Z = -236.768  mm,
	W = 0.000 deg,	P = 30.000 deg,	R = 178.417 deg
};
P[320]{
   GP1:
	UF : 0, UT : 1,		CONFIG : 'N U T, 0, 0, 0',
	X = 1221.024  mm,	Y = 137.193  mm,	Z = -236.746  mm,
	W = 0.000 deg,	P = 30.000 deg,	R = 178.417 deg
};
P[321]{
   GP1:
	UF : 0, UT : 1,		CONFIG : 'N U T, 0, 0, 0',
	X = 1221.079  mm,	Y = 139.192  mm,	Z = -236.724  mm,
	W = 0.000 deg,	P = 30.000 deg,	R = 178.417 deg
};
P[322]{
   GP1:
	UF : 0, UT : 1,		CONFIG : 'N U T, 0, 0, 0',
	X = 1211.138  mm,	Y = 141.468  mm,	Z = -236.702  mm,
	W = 0.000 deg,	P = 30.000 deg,	R = 178.417 deg
};
P[323]{
   GP1:
	UF : 0, UT : 1,		CONFIG : 'N U T, 0, 0, 0',
	X = 1211.194  mm,	Y = 143.467  mm,	Z = -236.680  mm,
	W = 0.000 deg,	P = 30.000 deg,	R = 178.417 deg
};
P[324]{
   GP1:
	UF : 0, UT : 1,		CONFIG : 'N U T, 0, 0, 0',
	X = 1221.245  mm,	Y = 145.189  mm,	Z = -236.658  mm,
	W = 0.000 deg,	P = 30.000 deg,	R = 178.417 deg
};
P[325]{
   GP1:
	UF : 0, UT : 1,		CONFIG : 'N U T, 0, 0, 0',
	X = 1221.300  mm,	Y = 147.189  mm,	Z = -236.636  mm,
	W = 0.000 deg,	P = 30.000 deg,	R = 178.417 deg
};
P[326]{
   GP1:
	UF : 0, UT : 1,		CONFIG : 'N U T, 0, 0, 0',
	X = 1221.356  mm,	Y = 149.188  mm,	Z = -236.614  mm,
	W = 0.000 deg,	P = 30.000 deg,	R = 178.417 deg
};
P[327]{
   GP1:
	UF : 0, UT : 1,		CONFIG : 'N U T, 0, 0, 0',
	X = 1221.411  mm,	Y = 151.187  mm,	Z = -236.592  mm,
	W = 0.000 deg,	P = 30.000 deg,	R = 178.417 deg
};
P[328]{
   GP1:
	UF : 0, UT : 1,		CONFIG : 'N U T, 0, 0, 0',
	X = 1211.470  mm,	Y = 153.462  mm,	Z = -236.570  mm,
	W = 0.000 deg,	P = 30.000 deg,	R = 178.417 deg
};
P[329]{
   GP1:
	UF : 0, UT : 1,		CONFIG : 'N U T, 0, 0, 0',
	X = 1211.525  mm,	Y = 155.461  mm,	Z = -236.548  mm,
	W = 0.000 deg,	P = 30.000 deg,	R = 178.417 deg
};
P[330]{
   GP1:
	UF : 0, UT : 1,		CONFIG : 'N U T, 0, 0, 0',
	X = 1221.577  mm,	Y = 157.184  mm,	Z = -236.526  mm,
	W = 0.000 deg,	P = 30.000 deg,	R = 178.417 deg
};
P[331]{
   GP1:
	UF : 0, UT : 1,		CONFIG : 'N U T, 0, 0, 0',
	X = 1221.632  mm,	Y = 159.183  mm,	Z = -236.504  mm,
	W = 0.000 deg,	P = 30.000 deg,	R = 178.417 deg
};
P[332]{
   GP1:
	UF : 0, UT : 1,		CONFIG : 'N U T, 0, 0, 0',
	X = 1221.687  mm,	Y = 161.182  mm,	Z = -236.482  mm,
	W = 0.000 deg,	P = 30.000 deg,	R = 178.417 deg
};
P[333]{
   GP1:
	UF : 0, UT : 1,		CONFIG : 'N U T, 0, 0, 0',
	X = 1221.742  mm,	Y = 163.182  mm,	Z = -236.460  mm,
	W = 0.000 deg,	P = 30.000 deg,	R = 178.417 deg
};
P[334]{
   GP1:
	UF : 0, UT : 1,		CONFIG : 'N U T, 0, 0, 0',
	X = 1211.802  mm,	Y = 165.457  mm,	Z = -236.438  mm,
	W = 0.000 deg,	P = 30.000 deg,	R = 176.928 deg
};
P[335]{
   GP1:
	UF : 0, UT : 1,		CONFIG : 'N U T, 0, 0, 0',
	X = 1211.857  mm,	Y = 167.456  mm,	Z = -236.416  mm,
	W = 0.000 deg,	P = 30.000 deg,	R = 168.346 deg
};
P[336]{
   GP1:
	UF : 0, UT : 1,		CONFIG : 'N U T, 0, 0, 0',
	X = 1211.912  mm,	Y = 169.455  mm,	Z = -236.394  mm,
	W = 0.000 deg,	P = 30.000 deg,	R = 159.764 deg
};
P[337]{
   GP1:
	UF : 0, UT : 1,		CONFIG : 'N U T, 0, 0, 0',
	X = 1211.967  mm,	Y = 171.454  mm,	Z = -236.372  mm,
	W = 0.000 deg,	P = 30.000 deg,	R = 151.182 deg
};
P[338]{
   GP1:
	UF : 0, UT : 1,		CONFIG : 'N U T, 0, 0, 0',
	X = 1212.023  mm,	Y = 173.453  mm,	Z = -236.350  mm,
	W = 0.000 deg,	P = 30.000 deg,	R = 142.599 deg
};
P[339]{
   GP1:
	UF : 0, UT : 1,		CONFIG : 'N U T, 0, 0, 0',
	X = 1212.080  mm,	Y = 175.490  mm,	Z = -236.328  mm,
	W = 0.000 deg,	P = 30.000 deg,	R = 135.506 deg
};
P[340]{
   GP1:
	UF : 0, UT : 1,		CONFIG : 'N U T, 0, 0, 0',
	X = 1220.679  mm,	Y = 171.794  mm,	Z = -236.336  mm,
	W = 0.000 deg,	P = 30.000 deg,	R = 135.506 deg
};
P[341]{
   GP1:
	UF : 0, UT : 1,		CONFIG : 'N U T, 0, 0, 0',
	X = 1222.066  mm,	Y = 173.206  mm,	Z = -236.622  mm,
	W = 0.000 deg,	P = 30.000 deg,	R = 135.506 deg
};
P[342]{
   GP1:
	UF : 0, UT : 1,		CONFIG : 'N U T, 0, 0, 0',
	X = 1223.453  mm,	Y = 174.618  mm,	Z = -236.908  mm,
	W = 0.000 deg,	P = 30.000 deg,	R = 135.506 deg
};
P[343]{
   GP1:
	UF : 0, UT : 1,		CONFIG : 'N U T, 0, 0, 0',
	X = 1217.707  mm,	Y = 183.039  mm,	Z = -237.193  mm,
	W = 0.000 deg,	P = 30.000 deg,	R = 135.506 deg
};
P[344]{
   GP1:
	UF : 0, UT : 1,		CONFIG : 'N U T, 0, 0, 0',
	X = 1226.228  mm,	Y = 177.442  mm,	Z = -237.479  mm,
	W = 0.000 deg,	P = 30.000 deg,	R = 135.506 deg
};
P[345]{
   GP1:
	UF : 0, UT : 1,		CONFIG : 'N U T, 0, 0, 0',
	X = 1227.615  mm,	Y = 178.854  mm,	Z = -237.765  mm,
	W = 0.000 deg,	P = 30.000 deg,	R = 135.506 deg
};
P[346]{
   GP1:
	UF : 0, UT : 1,		CONFIG : 'N U T, 0, 0, 0',
	X = 1229.002  mm,	Y = 180.266  mm,	Z = -238.050  mm,
	W = 0.000 deg,	P = 30.000 deg,	R = 135.506 deg
};
P[347]{
   GP1:
	UF : 0, UT : 1,		CONFIG : 'N U T, 0, 0, 0',
	X = 1230.390  mm,	Y = 181.678  mm,	Z = -238.336  mm,
	W = 0.000 deg,	P = 30.000 deg,	R = 135.506 deg
};
P[348]{
   GP1:
	UF : 0, UT : 1,		CONFIG : 'N U T, 0, 0, 0',
	X = 1224.644  mm,	Y = 190.099  mm,	Z = -238.622  mm,
	W = 0.000 deg,	P = 30.000 deg,	R = 135.506 deg
};
P[349]{
   GP1:
	UF : 0, UT : 1,		CONFIG : 'N U T, 0, 0, 0',
	X = 1233.164  mm,	Y = 184.502  mm,	Z = -238.908  mm,
	W = 0.000 deg,	P = 30.000 deg,	R = 135.506 deg
};
P[350]{
   GP1:
	UF : 0, UT : 1,		CONFIG : 'N U T, 0, 0, 0',
	X = 1234.551  mm,	Y = 185.914  mm,	Z = -239.193  mm,
	W = 0.000 deg,	P = 30.000 deg,	R = 135.506 deg
};
P[351]{
   GP1:
	UF : 0, UT : 1,		CONFIG : 'N U T, 0, 0, 0',
	X = 1228.806  mm,	Y = 194.335  mm,	Z = -239.479  mm,
	W = 0.000 deg,	P = 30.000 deg,	R = 135.506 deg
};
P[352]{
   GP1:
	UF : 0, UT : 1,		CONFIG : 'N U T, 0, 0, 0',
	X = 1230.193  mm,	Y = 195.747  mm,	Z = -239.765  mm,
	W = 0.000 deg,	P = 30.000 deg,	R = 135.506 deg
};
P[353]{
   GP1:
	UF : 0, UT : 1,		CONFIG : 'N U T, 0, 0, 0',
	X = 1238.713  mm,	Y = 190.150  mm,	Z = -240.051  mm,
	W = 0.000 deg,	P = 30.000 deg,	R = 135.506 deg
};
P[354]{
   GP1:
	UF : 0, UT : 1,		CONFIG : 'N U T, 0, 0, 0',
	X = 1240.101  mm,	Y = 191.562  mm,	Z = -240.336  mm,
	W = 0.000 deg,	P = 30.000 deg,	R = 135.506 deg
};
P[355]{
   GP1:
	UF : 0, UT : 1,		CONFIG : 'N U T, 0, 0, 0',
	X = 1234.355  mm,	Y = 199.983  mm,	Z = -240.622  mm,
	W = 0.000 deg,	P = 30.000 deg,	R = 135.506 deg
};
P[356]{
   GP1:
	UF : 0, UT : 1,		CONFIG : 'N U T, 0, 0, 0',
	X = 1242.875  mm,	Y = 194.386  mm,	Z = -240.908  mm,
	W = 0.000 deg,	P = 30.000 deg,	R = 135.506 deg
};
P[357]{
   GP1:
	UF : 0, UT : 1,		CONFIG : 'N U T, 0, 0, 0',
	X = 1244.263  mm,	Y = 195.798  mm,	Z = -241.193  mm,
	W = 0.000 deg,	P = 30.000 deg,	R = 135.506 deg
};
P[358]{
   GP1:
	UF : 0, UT : 1,		CONFIG : 'N U T, 0, 0, 0',
	X = 1245.650  mm,	Y = 197.210  mm,	Z = -241.479  mm,
	W = 0.000 deg,	P = 30.000 deg,	R = 135.506 deg
};
P[359]{
   GP1:
	UF : 0, UT : 1,		CONFIG : 'N U T, 0, 0, 0',
	X = 1247.037  mm,	Y = 198.622  mm,	Z = -241.765  mm,
	W = 0.000 deg,	P = 30.000 deg,	R = 135.506 deg
};
P[360]{
   GP1:
	UF : 0, UT : 1,		CONFIG : 'N U T, 0, 0, 0',
	X = 1241.291  mm,	Y = 207.043  mm,	Z = -242.051  mm,
	W = 0.000 deg,	P = 30.000 deg,	R = 135.506 deg
};
P[361]{
   GP1:
	UF : 0, UT : 1,		CONFIG : 'N U T, 0, 0, 0',
	X = 1249.812  mm,	Y = 201.447  mm,	Z = -242.336  mm,
	W = 0.000 deg,	P = 30.000 deg,	R = 144.495 deg
};
P[362]{
   GP1:
	UF : 0, UT : 1,		CONFIG : 'N U T, 0, 0, 0',
	X = 1251.199  mm,	Y = 202.859  mm,	Z = -242.622  mm,
	W = 0.000 deg,	P = 30.000 deg,	R = 153.247 deg
};
P[363]{
   GP1:
	UF : 0, UT : 1,		CONFIG : 'N U T, 0, 0, 0',
	X = 1252.586  mm,	Y = 204.271  mm,	Z = -242.908  mm,
	W = 0.000 deg,	P = 30.000 deg,	R = 161.999 deg
};
P[364]{
   GP1:
	UF : 0, UT : 1,		CONFIG : 'N U T, 0, 0, 0',
	X = 1253.974  mm,	Y = 205.683  mm,	Z = -243.193  mm,
	W = 0.000 deg,	P = 30.000 deg,	R = 170.752 deg
};
P[365]{
   GP1:
	UF : 0, UT : 1,		CONFIG : 'N U T, 0, 0, 0',
	X = 1255.361  mm,	Y = 207.095  mm,	Z = -243.479  mm,
	W = 0.000 deg,	P = 30.000 deg,	R = 179.267 deg
};
P[366]{
   GP1:
	UF : 0, UT : 1,		CONFIG : 'N U T, 0, 0, 0',
	X = 1257.108  mm,	Y = 209.394  mm,	Z = -243.622  mm,
	W = 0.000 deg,	P = 30.000 deg,	R = 179.267 deg
};
P[367]{
   GP1:
	UF : 0, UT : 1,		CONFIG : 'N U T, 0, 0, 0',
	X = 1257.499  mm,	Y = 212.241  mm,	Z = -243.613  mm,
	W = 0.000 deg,	P = 30.000 deg,	R = 179.267 deg
};
P[368]{
   GP1:
	UF : 0, UT : 1,		CONFIG : 'N U T, 0, 0, 0',
	X = 1257.524  mm,	Y = 214.241  mm,	Z = -243.595  mm,
	W = 0.000 deg,	P = 30.000 deg,	R = 179.267 deg
};
P[369]{
   GP1:
	UF : 0, UT : 1,		CONFIG : 'N U T, 0, 0, 0',
	X = 1257.550  mm,	Y = 216.241  mm,	Z = -243.578  mm,
	W = 0.000 deg,	P = 30.000 deg,	R = 179.267 deg
};
P[370]{
   GP1:
	UF : 0, UT : 1,		CONFIG : 'N U T, 0, 0, 0',
	X = 1257.576  mm,	Y = 218.241  mm,	Z = -243.560  mm,
	W = 0.000 deg,	P = 30.000 deg,	R = 179.267 deg
};
P[371]{
   GP1:
	UF : 0, UT : 1,		CONFIG : 'N U T, 0, 0, 0',
	X = 1257.601  mm,	Y = 220.240  mm,	Z = -243.542  mm,
	W = 0.000 deg,	P = 30.000 deg,	R = 179.267 deg
};
P[372]{
   GP1:
	UF : 0, UT : 1,		CONFIG : 'N U T, 0, 0, 0',
	X = 1257.627  mm,	Y = 222.240  mm,	Z = -243.524  mm,
	W = 0.000 deg,	P = 30.000 deg,	R = 179.267 deg
};
P[373]{
   GP1:
	UF : 0, UT : 1,		CONFIG : 'N U T, 0, 0, 0',
	X = 1257.652  mm,	Y = 224.240  mm,	Z = -243.507  mm,
	W = 0.000 deg,	P = 30.000 deg,	R = 179.267 deg
};
P[374]{
   GP1:
	UF : 0, UT : 1,		CONFIG : 'N U T, 0, 0, 0',
	X = 1257.678  mm,	Y = 226.240  mm,	Z = -243.489  mm,
	W = 0.000 deg,	P = 30.000 deg,	R = 179.267 deg
};
P[375]{
   GP1:
	UF : 0, UT : 1,		CONFIG : 'N U T, 0, 0, 0',
	X = 1247.704  mm,	Y = 228.367  mm,	Z = -243.471  mm,
	W = 0.000 deg,	P = 30.000 deg,	R = 179.267 deg
};
P[376]{
   GP1:
	UF : 0, UT : 1,		CONFIG : 'N U T, 0, 0, 0',
	X = 1247.717  mm,	Y = 229.365  mm,	Z = -243.463  mm,
	W = 0.000 deg,	P = 30.000 deg,	R = 179.267 deg
};
/END
